Fanuc TP program (LS listing): hs0301h80_3.ls

/PROG  hs0301h80_3
/ATTR
COMMENT	= "19-03-01 11:47:14";
PROG_SIZE	= 0;
DEFAULT_GROUP	= 1, *, *, *, *;
/APPL
    ARC Welding Equipment: 1, *, *, *, *;
/MN
   1:  CALL HOME_ALL;
   1:  UFRAME_NUM = 1;
   1:  UTOOL_NUM = 3;
   1:  COL GUARD ADJUST 150;
   1:  PR[91] = PR[90];
   1:  PR[91,1] = PR[90,1] + -0.293;
   1:  PR[91,2] = PR[90,2] + 23.494;
   1:  PR[91,3] = PR[90,3] + 60.085;
   1:  PR[92] = PR[91];
   1:  PR[92,3] = PR[92,3] + 50;
   1:J PR[92] 10% FINE;
   1:L PR[91] R[100]mm/sec CNT100;
   1:  CALL LASER_DRAHT_START;
   1:  PR[91,1] = PR[90,1] + -6.009;
   1:  PR[91,2] = PR[90,2] + 23.979;
   1:L PR[91] R[100]mm/sec CNT100;
   1:  PR[91,1] = PR[90,1] + -6.508;
   1:  PR[91,2] = PR[90,2] + 23.917;
   1:L PR[91] R[100]mm/sec CNT100;
   1:  PR[91,1] = PR[90,1] + -12.344;
   1:  PR[91,2] = PR[90,2] + 22.945;
   1:L PR[91] R[100]mm/sec CNT100;
   1:  PR[91,1] = PR[90,1] + -12.597;
   1:  PR[91,2] = PR[90,2] + 22.847;
   1:L PR[91] R[100]mm/sec CNT100;
   1:  PR[91,1] = PR[90,1] + -18.195;
   1:  PR[91,2] = PR[90,2] + 20.363;
   1:L PR[91] R[100]mm/sec CNT100;
   1:  PR[91,1] = PR[90,1] + -18.230;
   1:  PR[91,2] = PR[90,2] + 20.339;
   1:L PR[91] R[100]mm/sec CNT100;
   1:  PR[91,1] = PR[90,1] + -23.139;
   1:  PR[91,2] = PR[90,2] + 16.449;
   1:L PR[91] R[100]mm/sec CNT100;
   1:  PR[91,1] = PR[90,1] + -26.912;
   1:  PR[91,2] = PR[90,2] + 11.480;
   1:L PR[91] R[100]mm/sec CNT100;
   1:  PR[91,1] = PR[90,1] + -29.270;
   1:  PR[91,2] = PR[90,2] + 5.788;
   1:L PR[91] R[100]mm/sec CNT100;
   1:  PR[91,1] = PR[90,1] + -30.068;
   1:  PR[91,2] = PR[90,2] + -0.337;
   1:L PR[91] R[100]mm/sec CNT100;
   1:  PR[91,1] = PR[90,1] + -30.060;
   1:  PR[91,2] = PR[90,2] + -0.419;
   1:L PR[91] R[100]mm/sec CNT100;
   1:  PR[91,1] = PR[90,1] + -29.269;
   1:  PR[91,2] = PR[90,2] + -6.417;
   1:L PR[91] R[100]mm/sec CNT100;
   1:  PR[91,1] = PR[90,1] + -26.906;
   1:  PR[91,2] = PR[90,2] + -12.115;
   1:L PR[91] R[100]mm/sec CNT100;
   1:  PR[91,1] = PR[90,1] + -23.137;
   1:  PR[91,2] = PR[90,2] + -17.075;
   1:L PR[91] R[100]mm/sec CNT100;
   1:  PR[91,1] = PR[90,1] + -18.184;
   1:  PR[91,2] = PR[90,2] + -20.996;
   1:L PR[91] R[100]mm/sec CNT100;
   1:  PR[91,1] = PR[90,1] + -12.564;
   1:  PR[91,2] = PR[90,2] + -23.482;
   1:L PR[91] R[100]mm/sec CNT100;
   1:  PR[91,1] = PR[90,1] + -12.309;
   1:  PR[91,2] = PR[90,2] + -23.579;
   1:L PR[91] R[100]mm/sec CNT100;
   1:  PR[91,1] = PR[90,1] + -6.470;
   1:  PR[91,2] = PR[90,2] + -24.544;
   1:L PR[91] R[100]mm/sec CNT100;
   1:  PR[91,1] = PR[90,1] + -5.966;
   1:  PR[91,2] = PR[90,2] + -24.604;
   1:L PR[91] R[100]mm/sec CNT100;
   1:  PR[91,1] = PR[90,1] + -0.295;
   1:  PR[91,2] = PR[90,2] + -24.113;
   1:L PR[91] R[100]mm/sec CNT100;
   1:  PR[91,1] = PR[90,1] + 0.454;
   1:  PR[91,2] = PR[90,2] + -24.114;
   1:L PR[91] R[100]mm/sec CNT100;
   1:  PR[91,1] = PR[90,1] + 5.405;
   1:  PR[91,2] = PR[90,2] + -24.549;
   1:L PR[91] R[100]mm/sec CNT100;
   1:  PR[91,1] = PR[90,1] + 6.160;
   1:  PR[91,2] = PR[90,2] + -24.608;
   1:L PR[91] R[100]mm/sec CNT100;
   1:  PR[91,1] = PR[90,1] + 6.349;
   1:  PR[91,2] = PR[90,2] + -24.596;
   1:L PR[91] R[100]mm/sec CNT100;
   1:  PR[91,1] = PR[90,1] + 12.478;
   1:  PR[91,2] = PR[90,2] + -23.575;
   1:L PR[91] R[100]mm/sec CNT100;
   1:  PR[91,1] = PR[90,1] + 12.730;
   1:  PR[91,2] = PR[90,2] + -23.477;
   1:L PR[91] R[100]mm/sec CNT100;
   1:  PR[91,1] = PR[90,1] + 18.333;
   1:  PR[91,2] = PR[90,2] + -20.999;
   1:L PR[91] R[100]mm/sec CNT100;
   1:  PR[91,1] = PR[90,1] + 18.368;
   1:  PR[91,2] = PR[90,2] + -20.974;
   1:L PR[91] R[100]mm/sec CNT100;
   1:  PR[91,1] = PR[90,1] + 23.284;
   1:  PR[91,2] = PR[90,2] + -17.085;
   1:L PR[91] R[100]mm/sec CNT100;
   1:  PR[91,1] = PR[90,1] + 27.064;
   1:  PR[91,2] = PR[90,2] + -12.111;
   1:L PR[91] R[100]mm/sec CNT100;
   1:  PR[91,1] = PR[90,1] + 29.425;
   1:  PR[91,2] = PR[90,2] + -6.423;
   1:L PR[91] R[100]mm/sec CNT100;
   1:  PR[91,1] = PR[90,1] + 30.225;
   1:  PR[91,2] = PR[90,2] + -0.287;
   1:L PR[91] R[100]mm/sec CNT100;
   1:  PR[91,1] = PR[90,1] + 30.217;
   1:  PR[91,2] = PR[90,2] + -0.204;
   1:L PR[91] R[100]mm/sec CNT100;
   1:  PR[91,1] = PR[90,1] + 29.427;
   1:  PR[91,2] = PR[90,2] + 5.793;
   1:L PR[91] R[100]mm/sec CNT100;
   1:  PR[91,1] = PR[90,1] + 27.069;
   1:  PR[91,2] = PR[90,2] + 11.477;
   1:L PR[91] R[100]mm/sec CNT100;
   1:  PR[91,1] = PR[90,1] + 23.297;
   1:  PR[91,2] = PR[90,2] + 16.449;
   1:L PR[91] R[100]mm/sec CNT100;
   1:  PR[91,1] = PR[90,1] + 18.388;
   1:  PR[91,2] = PR[90,2] + 20.339;
   1:L PR[91] R[100]mm/sec CNT100;
   1:  PR[91,1] = PR[90,1] + 18.353;
   1:  PR[91,2] = PR[90,2] + 20.363;
   1:L PR[91] R[100]mm/sec CNT100;
   1:  PR[91,1] = PR[90,1] + 12.755;
   1:  PR[91,2] = PR[90,2] + 22.846;
   1:L PR[91] R[100]mm/sec CNT100;
   1:  PR[91,1] = PR[90,1] + 12.502;
   1:  PR[91,2] = PR[90,2] + 22.944;
   1:L PR[91] R[100]mm/sec CNT100;
   1:  PR[91,1] = PR[90,1] + 6.667;
   1:  PR[91,2] = PR[90,2] + 23.917;
   1:L PR[91] R[100]mm/sec CNT100;
   1:  PR[91,1] = PR[90,1] + 6.167;
   1:  PR[91,2] = PR[90,2] + 23.979;
   1:L PR[91] R[100]mm/sec CNT100;
   1:  PR[91,1] = PR[90,1] + 0.451;
   1:  PR[91,2] = PR[90,2] + 23.494;
   1:L PR[91] R[100]mm/sec CNT100;
   1:  PR[91] = PR[90];
   1:  PR[91,1] = PR[90,1] + -0.281;
   1:  PR[91,2] = PR[90,2] + 23.657;
   1:  PR[91,3] = PR[90,3] + 60.695;
   1:L PR[91] R[100]mm/sec CNT100;
   1:  PR[91,1] = PR[90,1] + -3.910;
   1:  PR[91,2] = PR[90,2] + 23.972;
   1:L PR[91] R[100]mm/sec CNT100;
   1:  PR[91,1] = PR[90,1] + -5.747;
   1:  PR[91,2] = PR[90,2] + 24.117;
   1:L PR[91] R[100]mm/sec CNT100;
   1:  PR[91,1] = PR[90,1] + -6.520;
   1:  PR[91,2] = PR[90,2] + 24.021;
   1:L PR[91] R[100]mm/sec CNT100;
   1:  PR[91,1] = PR[90,1] + -12.103;
   1:  PR[91,2] = PR[90,2] + 23.091;
   1:L PR[91] R[100]mm/sec CNT100;
   1:  PR[91,1] = PR[90,1] + -12.618;
   1:  PR[91,2] = PR[90,2] + 22.891;
   1:L PR[91] R[100]mm/sec CNT100;
   1:  PR[91,1] = PR[90,1] + -17.973;
   1:  PR[91,2] = PR[90,2] + 20.516;
   1:L PR[91] R[100]mm/sec CNT100;
   1:  PR[91,1] = PR[90,1] + -18.245;
   1:  PR[91,2] = PR[90,2] + 20.323;
   1:L PR[91] R[100]mm/sec CNT100;
   1:  PR[91,1] = PR[90,1] + -22.986;
   1:  PR[91,2] = PR[90,2] + 16.568;
   1:L PR[91] R[100]mm/sec CNT100;
   1:  PR[91,1] = PR[90,1] + -23.039;
   1:  PR[91,2] = PR[90,2] + 16.508;
   1:L PR[91] R[100]mm/sec CNT100;
   1:  PR[91,1] = PR[90,1] + -26.772;
   1:  PR[91,2] = PR[90,2] + 11.549;
   1:L PR[91] R[100]mm/sec CNT100;
   1:  PR[91,1] = PR[90,1] + -29.127;
   1:  PR[91,2] = PR[90,2] + 5.807;
   1:L PR[91] R[100]mm/sec CNT100;
   1:  PR[91,1] = PR[90,1] + -29.691;
   1:  PR[91,2] = PR[90,2] + 1.477;
   1:L PR[91] R[100]mm/sec CNT100;
   1:  PR[91,1] = PR[90,1] + -29.926;
   1:  PR[91,2] = PR[90,2] + -0.313;
   1:L PR[91] R[100]mm/sec CNT100;
   1:  PR[91,1] = PR[90,1] + -29.126;
   1:  PR[91,2] = PR[90,2] + -6.434;
   1:L PR[91] R[100]mm/sec CNT100;
   1:  PR[91,1] = PR[90,1] + -26.767;
   1:  PR[91,2] = PR[90,2] + -12.181;
   1:L PR[91] R[100]mm/sec CNT100;
   1:  PR[91,1] = PR[90,1] + -23.035;
   1:  PR[91,2] = PR[90,2] + -17.133;
   1:L PR[91] R[100]mm/sec CNT100;
   1:  PR[91,1] = PR[90,1] + -22.969;
   1:  PR[91,2] = PR[90,2] + -17.208;
   1:L PR[91] R[100]mm/sec CNT100;
   1:  PR[91,1] = PR[90,1] + -18.054;
   1:  PR[91,2] = PR[90,2] + -21.096;
   1:L PR[91] R[100]mm/sec CNT100;
   1:  PR[91,1] = PR[90,1] + -17.983;
   1:  PR[91,2] = PR[90,2] + -21.140;
   1:L PR[91] R[100]mm/sec CNT100;
   1:  PR[91,1] = PR[90,1] + -12.579;
   1:  PR[91,2] = PR[90,2] + -23.531;
   1:L PR[91] R[100]mm/sec CNT100;
   1:  PR[91,1] = PR[90,1] + -12.060;
   1:  PR[91,2] = PR[90,2] + -23.726;
   1:L PR[91] R[100]mm/sec CNT100;
   1:  PR[91,1] = PR[90,1] + -6.479;
   1:  PR[91,2] = PR[90,2] + -24.649;
   1:L PR[91] R[100]mm/sec CNT100;
   1:  PR[91,1] = PR[90,1] + -5.703;
   1:  PR[91,2] = PR[90,2] + -24.741;
   1:L PR[91] R[100]mm/sec CNT100;
   1:  PR[91,1] = PR[90,1] + -0.280;
   1:  PR[91,2] = PR[90,2] + -24.276;
   1:L PR[91] R[100]mm/sec CNT100;
   1:  PR[91,1] = PR[90,1] + 0.438;
   1:L PR[91] R[100]mm/sec CNT100;
   1:  PR[91,1] = PR[90,1] + 5.904;
   1:  PR[91,2] = PR[90,2] + -24.744;
   1:L PR[91] R[100]mm/sec CNT100;
   1:  PR[91,1] = PR[90,1] + 6.232;
   1:  PR[91,2] = PR[90,2] + -24.725;
   1:L PR[91] R[100]mm/sec CNT100;
   1:  PR[91,1] = PR[90,1] + 11.997;
   1:  PR[91,2] = PR[90,2] + -23.769;
   1:L PR[91] R[100]mm/sec CNT100;
   1:  PR[91,1] = PR[90,1] + 12.226;
   1:  PR[91,2] = PR[90,2] + -23.725;
   1:L PR[91] R[100]mm/sec CNT100;
   1:  PR[91,1] = PR[90,1] + 12.754;
   1:  PR[91,2] = PR[90,2] + -23.520;
   1:L PR[91] R[100]mm/sec CNT100;
   1:  PR[91,1] = PR[90,1] + 18.112;
   1:  PR[91,2] = PR[90,2] + -21.151;
   1:L PR[91] R[100]mm/sec CNT100;
   1:  PR[91,1] = PR[90,1] + 18.385;
   1:  PR[91,2] = PR[90,2] + -20.958;
   1:L PR[91] R[100]mm/sec CNT100;
   1:  PR[91,1] = PR[90,1] + 23.131;
   1:  PR[91,2] = PR[90,2] + -17.203;
   1:L PR[91] R[100]mm/sec CNT100;
   1:  PR[91,1] = PR[90,1] + 23.184;
   1:  PR[91,2] = PR[90,2] + -17.144;
   1:L PR[91] R[100]mm/sec CNT100;
   1:  PR[91,1] = PR[90,1] + 26.923;
   1:  PR[91,2] = PR[90,2] + -12.181;
   1:L PR[91] R[100]mm/sec CNT100;
   1:  PR[91,1] = PR[90,1] + 29.283;
   1:  PR[91,2] = PR[90,2] + -6.442;
   1:L PR[91] R[100]mm/sec CNT100;
   1:  PR[91,1] = PR[90,1] + 30.083;
   1:  PR[91,2] = PR[90,2] + -0.312;
   1:L PR[91] R[100]mm/sec CNT100;
   1:  PR[91,1] = PR[90,1] + 29.285;
   1:  PR[91,2] = PR[90,2] + 5.810;
   1:L PR[91] R[100]mm/sec CNT100;
   1:  PR[91,1] = PR[90,1] + 26.930;
   1:  PR[91,2] = PR[90,2] + 11.544;
   1:L PR[91] R[100]mm/sec CNT100;
   1:  PR[91,1] = PR[90,1] + 23.204;
   1:  PR[91,2] = PR[90,2] + 16.496;
   1:L PR[91] R[100]mm/sec CNT100;
   1:  PR[91,1] = PR[90,1] + 23.139;
   1:  PR[91,2] = PR[90,2] + 16.570;
   1:L PR[91] R[100]mm/sec CNT100;
   1:  PR[91,1] = PR[90,1] + 18.403;
   1:  PR[91,2] = PR[90,2] + 20.323;
   1:L PR[91] R[100]mm/sec CNT100;
   1:  PR[91,1] = PR[90,1] + 18.131;
   1:  PR[91,2] = PR[90,2] + 20.516;
   1:L PR[91] R[100]mm/sec CNT100;
   1:  PR[91,1] = PR[90,1] + 12.776;
   1:  PR[91,2] = PR[90,2] + 22.891;
   1:L PR[91] R[100]mm/sec CNT100;
   1:  PR[91,1] = PR[90,1] + 12.261;
   1:  PR[91,2] = PR[90,2] + 23.090;
   1:L PR[91] R[100]mm/sec CNT100;
   1:  PR[91,1] = PR[90,1] + 6.678;
   1:  PR[91,2] = PR[90,2] + 24.021;
   1:L PR[91] R[100]mm/sec CNT100;
   1:  PR[91,1] = PR[90,1] + 5.905;
   1:  PR[91,2] = PR[90,2] + 24.117;
   1:L PR[91] R[100]mm/sec CNT100;
   1:  PR[91,1] = PR[90,1] + 4.068;
   1:  PR[91,2] = PR[90,2] + 23.972;
   1:L PR[91] R[100]mm/sec CNT100;
   1:  PR[91,1] = PR[90,1] + 0.438;
   1:  PR[91,2] = PR[90,2] + 23.657;
   1:L PR[91] R[100]mm/sec CNT100;
   1:  PR[91] = PR[90];
   1:  PR[91,1] = PR[90,1] + -0.266;
   1:  PR[91,2] = PR[90,2] + 23.820;
   1:  PR[91,3] = PR[90,3] + 61.305;
   1:L PR[91] R[100]mm/sec CNT100;
   1:  PR[91,1] = PR[90,1] + -3.087;
   1:  PR[91,2] = PR[90,2] + 24.065;
   1:L PR[91] R[100]mm/sec CNT100;
   1:  PR[91,1] = PR[90,1] + -5.489;
   1:  PR[91,2] = PR[90,2] + 24.255;
   1:L PR[91] R[100]mm/sec CNT100;
   1:  PR[91,1] = PR[90,1] + -6.532;
   1:  PR[91,2] = PR[90,2] + 24.126;
   1:L PR[91] R[100]mm/sec CNT100;
   1:  PR[91,1] = PR[90,1] + -11.861;
   1:  PR[91,2] = PR[90,2] + 23.237;
   1:L PR[91] R[100]mm/sec CNT100;
   1:  PR[91,1] = PR[90,1] + -12.639;
   1:  PR[91,2] = PR[90,2] + 22.936;
   1:L PR[91] R[100]mm/sec CNT100;
   1:  PR[91,1] = PR[90,1] + -17.751;
   1:  PR[91,2] = PR[90,2] + 20.668;
   1:L PR[91] R[100]mm/sec CNT100;
   1:  PR[91,1] = PR[90,1] + -18.261;
   1:  PR[91,2] = PR[90,2] + 20.307;
   1:L PR[91] R[100]mm/sec CNT100;
   1:  PR[91,1] = PR[90,1] + -22.787;
   1:  PR[91,2] = PR[90,2] + 16.722;
   1:L PR[91] R[100]mm/sec CNT100;
   1:  PR[91,1] = PR[90,1] + -23.006;
   1:  PR[91,2] = PR[90,2] + 16.476;
   1:L PR[91] R[100]mm/sec CNT100;
   1:  PR[91,1] = PR[90,1] + -26.589;
   1:  PR[91,2] = PR[90,2] + 11.717;
   1:L PR[91] R[100]mm/sec CNT100;
   1:  PR[91,1] = PR[90,1] + -26.683;
   1:  PR[91,2] = PR[90,2] + 11.554;
   1:L PR[91] R[100]mm/sec CNT100;
   1:  PR[91,1] = PR[90,1] + -28.980;
   1:  PR[91,2] = PR[90,2] + 5.964;
   1:L PR[91] R[100]mm/sec CNT100;
   1:  PR[91,1] = PR[90,1] + -29.019;
   1:  PR[91,2] = PR[90,2] + 5.848;
   1:L PR[91] R[100]mm/sec CNT100;
   1:  PR[91,1] = PR[90,1] + -29.815;
   1:  PR[91,2] = PR[90,2] + -0.312;
   1:L PR[91] R[100]mm/sec CNT100;
   1:  PR[91,1] = PR[90,1] + -29.020;
   1:  PR[91,2] = PR[90,2] + -6.471;
   1:L PR[91] R[100]mm/sec CNT100;
   1:  PR[91,1] = PR[90,1] + -28.986;
   1:  PR[91,2] = PR[90,2] + -6.576;
   1:L PR[91] R[100]mm/sec CNT100;
   1:  PR[91,1] = PR[90,1] + -26.690;
   1:  PR[91,2] = PR[90,2] + -12.163;
   1:L PR[91] R[100]mm/sec CNT100;
   1:  PR[91,1] = PR[90,1] + -26.592;
   1:  PR[91,2] = PR[90,2] + -12.338;
   1:L PR[91] R[100]mm/sec CNT100;
   1:  PR[91,1] = PR[90,1] + -23.014;
   1:  PR[91,2] = PR[90,2] + -17.084;
   1:L PR[91] R[100]mm/sec CNT100;
   1:  PR[91,1] = PR[90,1] + -22.771;
   1:  PR[91,2] = PR[90,2] + -17.361;
   1:L PR[91] R[100]mm/sec CNT100;
   1:  PR[91,1] = PR[90,1] + -17.951;
   1:  PR[91,2] = PR[90,2] + -21.175;
   1:L PR[91] R[100]mm/sec CNT100;
   1:  PR[91,1] = PR[90,1] + -17.752;
   1:  PR[91,2] = PR[90,2] + -21.296;
   1:L PR[91] R[100]mm/sec CNT100;
   1:  PR[91,1] = PR[90,1] + -12.593;
   1:  PR[91,2] = PR[90,2] + -23.579;
   1:L PR[91] R[100]mm/sec CNT100;
   1:  PR[91,1] = PR[90,1] + -11.812;
   1:  PR[91,2] = PR[90,2] + -23.874;
   1:L PR[91] R[100]mm/sec CNT100;
   1:  PR[91,1] = PR[90,1] + -6.489;
   1:  PR[91,2] = PR[90,2] + -24.754;
   1:L PR[91] R[100]mm/sec CNT100;
   1:  PR[91,1] = PR[90,1] + -5.435;
   1:  PR[91,2] = PR[90,2] + -24.879;
   1:L PR[91] R[100]mm/sec CNT100;
   1:  PR[91,1] = PR[90,1] + -4.039;
   1:  PR[91,2] = PR[90,2] + -24.770;
   1:L PR[91] R[100]mm/sec CNT100;
   1:  PR[91,1] = PR[90,1] + -0.268;
   1:  PR[91,2] = PR[90,2] + -24.438;
   1:L PR[91] R[100]mm/sec CNT100;
   1:  PR[91,1] = PR[90,1] + 0.425;
   1:L PR[91] R[100]mm/sec CNT100;
   1:  PR[91,1] = PR[90,1] + 4.197;
   1:  PR[91,2] = PR[90,2] + -24.770;
   1:L PR[91] R[100]mm/sec CNT100;
   1:  PR[91,1] = PR[90,1] + 5.636;
   1:  PR[91,2] = PR[90,2] + -24.882;
   1:L PR[91] R[100]mm/sec CNT100;
   1:  PR[91,1] = PR[90,1] + 6.114;
   1:  PR[91,2] = PR[90,2] + -24.853;
   1:L PR[91] R[100]mm/sec CNT100;
   1:  PR[91,1] = PR[90,1] + 11.615;
   1:  PR[91,2] = PR[90,2] + -23.941;
   1:L PR[91] R[100]mm/sec CNT100;
   1:  PR[91,1] = PR[90,1] + 11.989;
   1:  PR[91,2] = PR[90,2] + -23.870;
   1:L PR[91] R[100]mm/sec CNT100;
   1:  PR[91,1] = PR[90,1] + 12.777;
   1:  PR[91,2] = PR[90,2] + -23.564;
   1:L PR[91] R[100]mm/sec CNT100;
   1:  PR[91,1] = PR[90,1] + 17.890;
   1:  PR[91,2] = PR[90,2] + -21.303;
   1:L PR[91] R[100]mm/sec CNT100;
   1:  PR[91,1] = PR[90,1] + 18.401;
   1:  PR[91,2] = PR[90,2] + -20.941;
   1:L PR[91] R[100]mm/sec CNT100;
   1:  PR[91,1] = PR[90,1] + 22.933;
   1:  PR[91,2] = PR[90,2] + -17.357;
   1:L PR[91] R[100]mm/sec CNT100;
   1:  PR[91,1] = PR[90,1] + 23.152;
   1:  PR[91,2] = PR[90,2] + -17.111;
   1:L PR[91] R[100]mm/sec CNT100;
   1:  PR[91,1] = PR[90,1] + 26.740;
   1:  PR[91,2] = PR[90,2] + -12.348;
   1:L PR[91] R[100]mm/sec CNT100;
   1:  PR[91,1] = PR[90,1] + 26.835;
   1:  PR[91,2] = PR[90,2] + -12.185;
   1:L PR[91] R[100]mm/sec CNT100;
   1:  PR[91,1] = PR[90,1] + 29.135;
   1:  PR[91,2] = PR[90,2] + -6.598;
   1:L PR[91] R[100]mm/sec CNT100;
   1:  PR[91,1] = PR[90,1] + 29.174;
   1:  PR[91,2] = PR[90,2] + -6.482;
   1:L PR[91] R[100]mm/sec CNT100;
   1:  PR[91,1] = PR[90,1] + 29.965;
   1:  PR[91,2] = PR[90,2] + -0.403;
   1:L PR[91] R[100]mm/sec CNT100;
   1:  PR[91,1] = PR[90,1] + 29.974;
   1:  PR[91,2] = PR[90,2] + -0.325;
   1:L PR[91] R[100]mm/sec CNT100;
   1:  PR[91,1] = PR[90,1] + 29.178;
   1:  PR[91,2] = PR[90,2] + 5.846;
   1:L PR[91] R[100]mm/sec CNT100;
   1:  PR[91,1] = PR[90,1] + 29.145;
   1:  PR[91,2] = PR[90,2] + 5.951;
   1:L PR[91] R[100]mm/sec CNT100;
   1:  PR[91,1] = PR[90,1] + 26.852;
   1:  PR[91,2] = PR[90,2] + 11.526;
   1:L PR[91] R[100]mm/sec CNT100;
   1:  PR[91,1] = PR[90,1] + 26.754;
   1:  PR[91,2] = PR[90,2] + 11.701;
   1:L PR[91] R[100]mm/sec CNT100;
   1:  PR[91,1] = PR[90,1] + 23.183;
   1:  PR[91,2] = PR[90,2] + 16.448;
   1:L PR[91] R[100]mm/sec CNT100;
   1:  PR[91,1] = PR[90,1] + 22.940;
   1:  PR[91,2] = PR[90,2] + 16.724;
   1:L PR[91] R[100]mm/sec CNT100;
   1:  PR[91,1] = PR[90,1] + 18.419;
   1:  PR[91,2] = PR[90,2] + 20.307;
   1:L PR[91] R[100]mm/sec CNT100;
   1:  PR[91,1] = PR[90,1] + 17.909;
   1:  PR[91,2] = PR[90,2] + 20.668;
   1:L PR[91] R[100]mm/sec CNT100;
   1:  PR[91,1] = PR[90,1] + 12.797;
   1:  PR[91,2] = PR[90,2] + 22.935;
   1:L PR[91] R[100]mm/sec CNT100;
   1:  PR[91,1] = PR[90,1] + 12.019;
   1:  PR[91,2] = PR[90,2] + 23.237;
   1:L PR[91] R[100]mm/sec CNT100;
   1:  PR[91,1] = PR[90,1] + 6.690;
   1:  PR[91,2] = PR[90,2] + 24.126;
   1:L PR[91] R[100]mm/sec CNT100;
   1:  PR[91,1] = PR[90,1] + 5.647;
   1:  PR[91,2] = PR[90,2] + 24.255;
   1:L PR[91] R[100]mm/sec CNT100;
   1:  PR[91,1] = PR[90,1] + 3.244;
   1:  PR[91,2] = PR[90,2] + 24.065;
   1:L PR[91] R[100]mm/sec CNT100;
   1:  PR[91,1] = PR[90,1] + 0.424;
   1:  PR[91,2] = PR[90,2] + 23.820;
   1:L PR[91] R[100]mm/sec CNT100;
   1:  PR[91] = PR[90];
   1:  PR[91,1] = PR[90,1] + -0.249;
   1:  PR[91,2] = PR[90,2] + 23.984;
   1:  PR[91,3] = PR[90,3] + 61.915;
   1:L PR[91] R[100]mm/sec CNT100;
   1:  PR[91,1] = PR[90,1] + -5.233;
   1:  PR[91,2] = PR[90,2] + 24.392;
   1:L PR[91] R[100]mm/sec CNT100;
   1:  PR[91,1] = PR[90,1] + -6.544;
   1:  PR[91,2] = PR[90,2] + 24.230;
   1:L PR[91] R[100]mm/sec CNT100;
   1:  PR[91,1] = PR[90,1] + -11.619;
   1:  PR[91,2] = PR[90,2] + 23.384;
   1:L PR[91] R[100]mm/sec CNT100;
   1:  PR[91,1] = PR[90,1] + -12.660;
   1:  PR[91,2] = PR[90,2] + 22.981;
   1:L PR[91] R[100]mm/sec CNT100;
   1:  PR[91,1] = PR[90,1] + -17.529;
   1:  PR[91,2] = PR[90,2] + 20.821;
   1:L PR[91] R[100]mm/sec CNT100;
   1:  PR[91,1] = PR[90,1] + -18.277;
   1:  PR[91,2] = PR[90,2] + 20.291;
   1:L PR[91] R[100]mm/sec CNT100;
   1:  PR[91,1] = PR[90,1] + -22.588;
   1:  PR[91,2] = PR[90,2] + 16.876;
   1:L PR[91] R[100]mm/sec CNT100;
   1:  PR[91,1] = PR[90,1] + -22.974;
   1:  PR[91,2] = PR[90,2] + 16.443;
   1:L PR[91] R[100]mm/sec CNT100;
   1:  PR[91,1] = PR[90,1] + -26.386;
   1:  PR[91,2] = PR[90,2] + 11.910;
   1:L PR[91] R[100]mm/sec CNT100;
   1:  PR[91,1] = PR[90,1] + -26.605;
   1:  PR[91,2] = PR[90,2] + 11.534;
   1:L PR[91] R[100]mm/sec CNT100;
   1:  PR[91,1] = PR[90,1] + -28.792;
   1:  PR[91,2] = PR[90,2] + 6.211;
   1:L PR[91] R[100]mm/sec CNT100;
   1:  PR[91,1] = PR[90,1] + -28.917;
   1:  PR[91,2] = PR[90,2] + 5.841;
   1:L PR[91] R[100]mm/sec CNT100;
   1:  PR[91,1] = PR[90,1] + -29.707;
   1:  PR[91,2] = PR[90,2] + -0.311;
   1:L PR[91] R[100]mm/sec CNT100;
   1:  PR[91,1] = PR[90,1] + -28.963;
   1:  PR[91,2] = PR[90,2] + -6.019;
   1:L PR[91] R[100]mm/sec CNT100;
   1:  PR[91,1] = PR[90,1] + -28.916;
   1:  PR[91,2] = PR[90,2] + -6.465;
   1:L PR[91] R[100]mm/sec CNT100;
   1:  PR[91,1] = PR[90,1] + -28.810;
   1:  PR[91,2] = PR[90,2] + -6.797;
   1:L PR[91] R[100]mm/sec CNT100;
   1:  PR[91,1] = PR[90,1] + -26.623;
   1:  PR[91,2] = PR[90,2] + -12.117;
   1:L PR[91] R[100]mm/sec CNT100;
   1:  PR[91,1] = PR[90,1] + -26.401;
   1:  PR[91,2] = PR[90,2] + -12.515;
   1:L PR[91] R[100]mm/sec CNT100;
   1:  PR[91,1] = PR[90,1] + -22.993;
   1:  PR[91,2] = PR[90,2] + -17.036;
   1:L PR[91] R[100]mm/sec CNT100;
   1:  PR[91,1] = PR[90,1] + -22.572;
   1:  PR[91,2] = PR[90,2] + -17.515;
   1:L PR[91] R[100]mm/sec CNT100;
   1:  PR[91,1] = PR[90,1] + -17.849;
   1:  PR[91,2] = PR[90,2] + -21.254;
   1:L PR[91] R[100]mm/sec CNT100;
   1:  PR[91,1] = PR[90,1] + -17.521;
   1:  PR[91,2] = PR[90,2] + -21.453;
   1:L PR[91] R[100]mm/sec CNT100;
   1:  PR[91,1] = PR[90,1] + -12.608;
   1:  PR[91,2] = PR[90,2] + -23.627;
   1:L PR[91] R[100]mm/sec CNT100;
   1:  PR[91,1] = PR[90,1] + -11.563;
   1:  PR[91,2] = PR[90,2] + -24.022;
   1:L PR[91] R[100]mm/sec CNT100;
   1:  PR[91,1] = PR[90,1] + -6.498;
   1:  PR[91,2] = PR[90,2] + -24.860;
   1:L PR[91] R[100]mm/sec CNT100;
   1:  PR[91,1] = PR[90,1] + -5.173;
   1:  PR[91,2] = PR[90,2] + -25.016;
   1:L PR[91] R[100]mm/sec CNT100;
   1:  PR[91,1] = PR[90,1] + -3.435;
   1:  PR[91,2] = PR[90,2] + -24.881;
   1:L PR[91] R[100]mm/sec CNT100;
   1:  PR[91,1] = PR[90,1] + -0.254;
   1:  PR[91,2] = PR[90,2] + -24.601;
   1:L PR[91] R[100]mm/sec CNT100;
   1:  PR[91,1] = PR[90,1] + 0.411;
   1:L PR[91] R[100]mm/sec CNT100;
   1:  PR[91,1] = PR[90,1] + 3.593;
   1:  PR[91,2] = PR[90,2] + -24.881;
   1:L PR[91] R[100]mm/sec CNT100;
   1:  PR[91,1] = PR[90,1] + 5.374;
   1:  PR[91,2] = PR[90,2] + -25.019;
   1:L PR[91] R[100]mm/sec CNT100;
   1:  PR[91,1] = PR[90,1] + 5.996;
   1:  PR[91,2] = PR[90,2] + -24.982;
   1:L PR[91] R[100]mm/sec CNT100;
   1:  PR[91,1] = PR[90,1] + 11.234;
   1:  PR[91,2] = PR[90,2] + -24.113;
   1:L PR[91] R[100]mm/sec CNT100;
   1:  PR[91,1] = PR[90,1] + 11.751;
   1:  PR[91,2] = PR[90,2] + -24.015;
   1:L PR[91] R[100]mm/sec CNT100;
   1:  PR[91,1] = PR[90,1] + 12.800;
   1:  PR[91,2] = PR[90,2] + -23.607;
   1:L PR[91] R[100]mm/sec CNT100;
   1:  PR[91,1] = PR[90,1] + 17.668;
   1:  PR[91,2] = PR[90,2] + -21.455;
   1:L PR[91] R[100]mm/sec CNT100;
   1:  PR[91,1] = PR[90,1] + 18.417;
   1:  PR[91,2] = PR[90,2] + -20.925;
   1:L PR[91] R[100]mm/sec CNT100;
   1:  PR[91,1] = PR[90,1] + 22.734;
   1:  PR[91,2] = PR[90,2] + -17.510;
   1:L PR[91] R[100]mm/sec CNT100;
   1:  PR[91,1] = PR[90,1] + 23.121;
   1:  PR[91,2] = PR[90,2] + -17.077;
   1:L PR[91] R[100]mm/sec CNT100;
   1:  PR[91,1] = PR[90,1] + 26.538;
   1:  PR[91,2] = PR[90,2] + -12.541;
   1:L PR[91] R[100]mm/sec CNT100;
   1:  PR[91,1] = PR[90,1] + 26.757;
   1:  PR[91,2] = PR[90,2] + -12.165;
   1:L PR[91] R[100]mm/sec CNT100;
   1:  PR[91,1] = PR[90,1] + 28.948;
   1:  PR[91,2] = PR[90,2] + -6.844;
   1:L PR[91] R[100]mm/sec CNT100;
   1:  PR[91,1] = PR[90,1] + 29.072;
   1:  PR[91,2] = PR[90,2] + -6.475;
   1:L PR[91] R[100]mm/sec CNT100;
   1:  PR[91,1] = PR[90,1] + 29.825;
   1:  PR[91,2] = PR[90,2] + -0.688;
   1:L PR[91] R[100]mm/sec CNT100;
   1:  PR[91,1] = PR[90,1] + 29.865;
   1:  PR[91,2] = PR[90,2] + -0.326;
   1:L PR[91] R[100]mm/sec CNT100;
   1:  PR[91,1] = PR[90,1] + 29.121;
   1:  PR[91,2] = PR[90,2] + 5.395;
   1:L PR[91] R[100]mm/sec CNT100;
   1:  PR[91,1] = PR[90,1] + 29.074;
   1:  PR[91,2] = PR[90,2] + 5.840;
   1:L PR[91] R[100]mm/sec CNT100;
   1:  PR[91,1] = PR[90,1] + 28.969;
   1:  PR[91,2] = PR[90,2] + 6.172;
   1:L PR[91] R[100]mm/sec CNT100;
   1:  PR[91,1] = PR[90,1] + 26.785;
   1:  PR[91,2] = PR[90,2] + 11.481;
   1:L PR[91] R[100]mm/sec CNT100;
   1:  PR[91,1] = PR[90,1] + 26.563;
   1:  PR[91,2] = PR[90,2] + 11.879;
   1:L PR[91] R[100]mm/sec CNT100;
   1:  PR[91,1] = PR[90,1] + 23.161;
   1:  PR[91,2] = PR[90,2] + 16.400;
   1:L PR[91] R[100]mm/sec CNT100;
   1:  PR[91,1] = PR[90,1] + 22.741;
   1:  PR[91,2] = PR[90,2] + 16.878;
   1:L PR[91] R[100]mm/sec CNT100;
   1:  PR[91,1] = PR[90,1] + 18.434;
   1:  PR[91,2] = PR[90,2] + 20.291;
   1:L PR[91] R[100]mm/sec CNT100;
   1:  PR[91,1] = PR[90,1] + 17.687;
   1:  PR[91,2] = PR[90,2] + 20.821;
   1:L PR[91] R[100]mm/sec CNT100;
   1:  PR[91,1] = PR[90,1] + 12.817;
   1:  PR[91,2] = PR[90,2] + 22.980;
   1:L PR[91] R[100]mm/sec CNT100;
   1:  PR[91,1] = PR[90,1] + 11.777;
   1:  PR[91,2] = PR[90,2] + 23.383;
   1:L PR[91] R[100]mm/sec CNT100;
   1:  PR[91,1] = PR[90,1] + 6.702;
   1:  PR[91,2] = PR[90,2] + 24.230;
   1:L PR[91] R[100]mm/sec CNT100;
   1:  PR[91,1] = PR[90,1] + 5.391;
   1:  PR[91,2] = PR[90,2] + 24.392;
   1:L PR[91] R[100]mm/sec CNT100;
   1:  PR[91,1] = PR[90,1] + 0.406;
   1:  PR[91,2] = PR[90,2] + 23.984;
   1:L PR[91] R[100]mm/sec CNT100;
   1:  PR[91] = PR[90];
   1:  PR[91,1] = PR[90,1] + -0.234;
   1:  PR[91,2] = PR[90,2] + 24.147;
   1:  PR[91,3] = PR[90,3] + 62.525;
   1:L PR[91] R[100]mm/sec CNT100;
   1:  PR[91,1] = PR[90,1] + -4.974;
   1:  PR[91,2] = PR[90,2] + 24.530;
   1:L PR[91] R[100]mm/sec CNT100;
   1:  PR[91,1] = PR[90,1] + -6.556;
   1:  PR[91,2] = PR[90,2] + 24.334;
   1:L PR[91] R[100]mm/sec CNT100;
   1:  PR[91,1] = PR[90,1] + -11.378;
   1:  PR[91,2] = PR[90,2] + 23.530;
   1:L PR[91] R[100]mm/sec CNT100;
   1:  PR[91,1] = PR[90,1] + -12.681;
   1:  PR[91,2] = PR[90,2] + 23.025;
   1:L PR[91] R[100]mm/sec CNT100;
   1:  PR[91,1] = PR[90,1] + -17.307;
   1:  PR[91,2] = PR[90,2] + 20.973;
   1:L PR[91] R[100]mm/sec CNT100;
   1:  PR[91,1] = PR[90,1] + -18.292;
   1:  PR[91,2] = PR[90,2] + 20.275;
   1:L PR[91] R[100]mm/sec CNT100;
   1:  PR[91,1] = PR[90,1] + -22.389;
   1:  PR[91,2] = PR[90,2] + 17.030;
   1:L PR[91] R[100]mm/sec CNT100;
   1:  PR[91,1] = PR[90,1] + -22.942;
   1:  PR[91,2] = PR[90,2] + 16.410;
   1:L PR[91] R[100]mm/sec CNT100;
   1:  PR[91,1] = PR[90,1] + -26.184;
   1:  PR[91,2] = PR[90,2] + 12.104;
   1:L PR[91] R[100]mm/sec CNT100;
   1:  PR[91,1] = PR[90,1] + -26.528;
   1:  PR[91,2] = PR[90,2] + 11.514;
   1:L PR[91] R[100]mm/sec CNT100;
   1:  PR[91,1] = PR[90,1] + -28.605;
   1:  PR[91,2] = PR[90,2] + 6.458;
   1:L PR[91] R[100]mm/sec CNT100;
   1:  PR[91,1] = PR[90,1] + -28.815;
   1:  PR[91,2] = PR[90,2] + 5.834;
   1:L PR[91] R[100]mm/sec CNT100;
   1:  PR[91,1] = PR[90,1] + -29.529;
   1:  PR[91,2] = PR[90,2] + 0.347;
   1:L PR[91] R[100]mm/sec CNT100;
   1:  PR[91,1] = PR[90,1] + -29.600;
   1:  PR[91,2] = PR[90,2] + -0.298;
   1:L PR[91] R[100]mm/sec CNT100;
   1:  PR[91,1] = PR[90,1] + -28.892;
   1:  PR[91,2] = PR[90,2] + -5.730;
   1:L PR[91] R[100]mm/sec CNT100;
   1:  PR[91,1] = PR[90,1] + -28.818;
   1:  PR[91,2] = PR[90,2] + -6.441;
   1:L PR[91] R[100]mm/sec CNT100;
   1:  PR[91,1] = PR[90,1] + -28.634;
   1:  PR[91,2] = PR[90,2] + -7.018;
   1:L PR[91] R[100]mm/sec CNT100;
   1:  PR[91,1] = PR[90,1] + -26.556;
   1:  PR[91,2] = PR[90,2] + -12.072;
   1:L PR[91] R[100]mm/sec CNT100;
   1:  PR[91,1] = PR[90,1] + -26.210;
   1:  PR[91,2] = PR[90,2] + -12.693;
   1:L PR[91] R[100]mm/sec CNT100;
   1:  PR[91,1] = PR[90,1] + -22.972;
   1:  PR[91,2] = PR[90,2] + -16.987;
   1:L PR[91] R[100]mm/sec CNT100;
   1:  PR[91,1] = PR[90,1] + -22.374;
   1:  PR[91,2] = PR[90,2] + -17.668;
   1:L PR[91] R[100]mm/sec CNT100;
   1:  PR[91,1] = PR[90,1] + -17.746;
   1:  PR[91,2] = PR[90,2] + -21.333;
   1:L PR[91] R[100]mm/sec CNT100;
   1:  PR[91,1] = PR[90,1] + -17.291;
   1:  PR[91,2] = PR[90,2] + -21.610;
   1:L PR[91] R[100]mm/sec CNT100;
   1:  PR[91,1] = PR[90,1] + -12.623;
   1:  PR[91,2] = PR[90,2] + -23.675;
   1:L PR[91] R[100]mm/sec CNT100;
   1:  PR[91,1] = PR[90,1] + -11.314;
   1:  PR[91,2] = PR[90,2] + -24.170;
   1:L PR[91] R[100]mm/sec CNT100;
   1:  PR[91,1] = PR[90,1] + -6.507;
   1:  PR[91,2] = PR[90,2] + -24.965;
   1:L PR[91] R[100]mm/sec CNT100;
   1:  PR[91,1] = PR[90,1] + -4.911;
   1:  PR[91,2] = PR[90,2] + -25.153;
   1:L PR[91] R[100]mm/sec CNT100;
   1:  PR[91,1] = PR[90,1] + -2.831;
   1:  PR[91,2] = PR[90,2] + -24.991;
   1:L PR[91] R[100]mm/sec CNT100;
   1:  PR[91,1] = PR[90,1] + -0.240;
   1:  PR[91,2] = PR[90,2] + -24.763;
   1:L PR[91] R[100]mm/sec CNT100;
   1:  PR[91,1] = PR[90,1] + 0.397;
   1:L PR[91] R[100]mm/sec CNT100;
   1:  PR[91,1] = PR[90,1] + 2.989;
   1:  PR[91,2] = PR[90,2] + -24.991;
   1:L PR[91] R[100]mm/sec CNT100;
   1:  PR[91,1] = PR[90,1] + 5.111;
   1:  PR[91,2] = PR[90,2] + -25.156;
   1:L PR[91] R[100]mm/sec CNT100;
   1:  PR[91,1] = PR[90,1] + 5.878;
   1:  PR[91,2] = PR[90,2] + -25.110;
   1:L PR[91] R[100]mm/sec CNT100;
   1:  PR[91,1] = PR[90,1] + 10.853;
   1:  PR[91,2] = PR[90,2] + -24.285;
   1:L PR[91] R[100]mm/sec CNT100;
   1:  PR[91,1] = PR[90,1] + 11.514;
   1:  PR[91,2] = PR[90,2] + -24.160;
   1:L PR[91] R[100]mm/sec CNT100;
   1:  PR[91,1] = PR[90,1] + 12.824;
   1:  PR[91,2] = PR[90,2] + -23.651;
   1:L PR[91] R[100]mm/sec CNT100;
   1:  PR[91,1] = PR[90,1] + 17.446;
   1:  PR[91,2] = PR[90,2] + -21.607;
   1:L PR[91] R[100]mm/sec CNT100;
   1:  PR[91,1] = PR[90,1] + 18.434;
   1:  PR[91,2] = PR[90,2] + -20.909;
   1:L PR[91] R[100]mm/sec CNT100;
   1:  PR[91,1] = PR[90,1] + 22.536;
   1:  PR[91,2] = PR[90,2] + -17.664;
   1:L PR[91] R[100]mm/sec CNT100;
   1:  PR[91,1] = PR[90,1] + 23.089;
   1:  PR[91,2] = PR[90,2] + -17.044;
   1:L PR[91] R[100]mm/sec CNT100;
   1:  PR[91,1] = PR[90,1] + 26.336;
   1:  PR[91,2] = PR[90,2] + -12.734;
   1:L PR[91] R[100]mm/sec CNT100;
   1:  PR[91,1] = PR[90,1] + 26.680;
   1:  PR[91,2] = PR[90,2] + -12.144;
   1:L PR[91] R[100]mm/sec CNT100;
   1:  PR[91,1] = PR[90,1] + 28.760;
   1:  PR[91,2] = PR[90,2] + -7.090;
   1:L PR[91] R[100]mm/sec CNT100;
   1:  PR[91,1] = PR[90,1] + 28.970;
   1:  PR[91,2] = PR[90,2] + -6.467;
   1:L PR[91] R[100]mm/sec CNT100;
   1:  PR[91,1] = PR[90,1] + 29.686;
   1:  PR[91,2] = PR[90,2] + -0.972;
   1:L PR[91] R[100]mm/sec CNT100;
   1:  PR[91,1] = PR[90,1] + 29.757;
   1:  PR[91,2] = PR[90,2] + -0.326;
   1:L PR[91] R[100]mm/sec CNT100;
   1:  PR[91,1] = PR[90,1] + 29.050;
   1:  PR[91,2] = PR[90,2] + 5.106;
   1:L PR[91] R[100]mm/sec CNT100;
   1:  PR[91,1] = PR[90,1] + 28.976;
   1:  PR[91,2] = PR[90,2] + 5.817;
   1:L PR[91] R[100]mm/sec CNT100;
   1:  PR[91,1] = PR[90,1] + 28.792;
   1:  PR[91,2] = PR[90,2] + 6.393;
   1:L PR[91] R[100]mm/sec CNT100;
   1:  PR[91,1] = PR[90,1] + 26.719;
   1:  PR[91,2] = PR[90,2] + 11.436;
   1:L PR[91] R[100]mm/sec CNT100;
   1:  PR[91,1] = PR[90,1] + 26.372;
   1:  PR[91,2] = PR[90,2] + 12.057;
   1:L PR[91] R[100]mm/sec CNT100;
   1:  PR[91,1] = PR[90,1] + 23.140;
   1:  PR[91,2] = PR[90,2] + 16.352;
   1:L PR[91] R[100]mm/sec CNT100;
   1:  PR[91,1] = PR[90,1] + 22.542;
   1:  PR[91,2] = PR[90,2] + 17.032;
   1:L PR[91] R[100]mm/sec CNT100;
   1:  PR[91,1] = PR[90,1] + 18.450;
   1:  PR[91,2] = PR[90,2] + 20.275;
   1:L PR[91] R[100]mm/sec CNT100;
   1:  PR[91,1] = PR[90,1] + 17.464;
   1:  PR[91,2] = PR[90,2] + 20.973;
   1:L PR[91] R[100]mm/sec CNT100;
   1:  PR[91,1] = PR[90,1] + 12.838;
   1:  PR[91,2] = PR[90,2] + 23.025;
   1:L PR[91] R[100]mm/sec CNT100;
   1:  PR[91,1] = PR[90,1] + 11.535;
   1:  PR[91,2] = PR[90,2] + 23.530;
   1:L PR[91] R[100]mm/sec CNT100;
   1:  PR[91,1] = PR[90,1] + 6.714;
   1:  PR[91,2] = PR[90,2] + 24.334;
   1:L PR[91] R[100]mm/sec CNT100;
   1:  PR[91,1] = PR[90,1] + 5.132;
   1:  PR[91,2] = PR[90,2] + 24.530;
   1:L PR[91] R[100]mm/sec CNT100;
   1:  PR[91,1] = PR[90,1] + 0.391;
   1:  PR[91,2] = PR[90,2] + 24.147;
   1:L PR[91] R[100]mm/sec CNT100;
   1:  PR[91] = PR[90];
   1:  PR[91,1] = PR[90,1] + -0.219;
   1:  PR[91,2] = PR[90,2] + 24.310;
   1:  PR[91,3] = PR[90,3] + 63.135;
   1:L PR[91] R[100]mm/sec CNT100;
   1:  PR[91,1] = PR[90,1] + -4.715;
   1:  PR[91,2] = PR[90,2] + 24.667;
   1:L PR[91] R[100]mm/sec CNT100;
   1:  PR[91,1] = PR[90,1] + -6.568;
   1:  PR[91,2] = PR[90,2] + 24.438;
   1:L PR[91] R[100]mm/sec CNT100;
   1:  PR[91,1] = PR[90,1] + -11.136;
   1:  PR[91,2] = PR[90,2] + 23.677;
   1:L PR[91] R[100]mm/sec CNT100;
   1:  PR[91,1] = PR[90,1] + -12.702;
   1:  PR[91,2] = PR[90,2] + 23.070;
   1:L PR[91] R[100]mm/sec CNT100;
   1:  PR[91,1] = PR[90,1] + -17.085;
   1:  PR[91,2] = PR[90,2] + 21.126;
   1:L PR[91] R[100]mm/sec CNT100;
   1:  PR[91,1] = PR[90,1] + -18.308;
   1:  PR[91,2] = PR[90,2] + 20.260;
   1:L PR[91] R[100]mm/sec CNT100;
   1:  PR[91,1] = PR[90,1] + -22.190;
   1:  PR[91,2] = PR[90,2] + 17.184;
   1:L PR[91] R[100]mm/sec CNT100;
   1:  PR[91,1] = PR[90,1] + -22.910;
   1:  PR[91,2] = PR[90,2] + 16.378;
   1:L PR[91] R[100]mm/sec CNT100;
   1:  PR[91,1] = PR[90,1] + -25.981;
   1:  PR[91,2] = PR[90,2] + 12.297;
   1:L PR[91] R[100]mm/sec CNT100;
   1:  PR[91,1] = PR[90,1] + -26.450;
   1:  PR[91,2] = PR[90,2] + 11.494;
   1:L PR[91] R[100]mm/sec CNT100;
   1:  PR[91,1] = PR[90,1] + -28.417;
   1:  PR[91,2] = PR[90,2] + 6.704;
   1:L PR[91] R[100]mm/sec CNT100;
   1:  PR[91,1] = PR[90,1] + -28.713;
   1:  PR[91,2] = PR[90,2] + 5.827;
   1:L PR[91] R[100]mm/sec CNT100;
   1:  PR[91,1] = PR[90,1] + -29.389;
   1:  PR[91,2] = PR[90,2] + 0.632;
   1:L PR[91] R[100]mm/sec CNT100;
   1:  PR[91,1] = PR[90,1] + -29.492;
   1:  PR[91,2] = PR[90,2] + -0.298;
   1:L PR[91] R[100]mm/sec CNT100;
   1:  PR[91,1] = PR[90,1] + -28.821;
   1:  PR[91,2] = PR[90,2] + -5.442;
   1:L PR[91] R[100]mm/sec CNT100;
   1:  PR[91,1] = PR[90,1] + -28.719;
   1:  PR[91,2] = PR[90,2] + -6.418;
   1:L PR[91] R[100]mm/sec CNT100;
   1:  PR[91,1] = PR[90,1] + -28.458;
   1:  PR[91,2] = PR[90,2] + -7.240;
   1:L PR[91] R[100]mm/sec CNT100;
   1:  PR[91,1] = PR[90,1] + -26.490;
   1:  PR[91,2] = PR[90,2] + -12.027;
   1:L PR[91] R[100]mm/sec CNT100;
   1:  PR[91,1] = PR[90,1] + -26.018;
   1:  PR[91,2] = PR[90,2] + -12.870;
   1:L PR[91] R[100]mm/sec CNT100;
   1:  PR[91,1] = PR[90,1] + -22.951;
   1:  PR[91,2] = PR[90,2] + -16.939;
   1:L PR[91] R[100]mm/sec CNT100;
   1:  PR[91,1] = PR[90,1] + -22.175;
   1:  PR[91,2] = PR[90,2] + -17.822;
   1:L PR[91] R[100]mm/sec CNT100;
   1:  PR[91,1] = PR[90,1] + -17.643;
   1:  PR[91,2] = PR[90,2] + -21.412;
   1:L PR[91] R[100]mm/sec CNT100;
   1:  PR[91,1] = PR[90,1] + -17.060;
   1:  PR[91,2] = PR[90,2] + -21.767;
   1:L PR[91] R[100]mm/sec CNT100;
   1:  PR[91,1] = PR[90,1] + -12.638;
   1:  PR[91,2] = PR[90,2] + -23.723;
   1:L PR[91] R[100]mm/sec CNT100;
   1:  PR[91,1] = PR[90,1] + -11.066;
   1:  PR[91,2] = PR[90,2] + -24.318;
   1:L PR[91] R[100]mm/sec CNT100;
   1:  PR[91,1] = PR[90,1] + -6.516;
   1:  PR[91,2] = PR[90,2] + -25.070;
   1:L PR[91] R[100]mm/sec CNT100;
   1:  PR[91,1] = PR[90,1] + -4.649;
   1:  PR[91,2] = PR[90,2] + -25.290;
   1:L PR[91] R[100]mm/sec CNT100;
   1:  PR[91,1] = PR[90,1] + -2.228;
   1:  PR[91,2] = PR[90,2] + -25.102;
   1:L PR[91] R[100]mm/sec CNT100;
   1:  PR[91,1] = PR[90,1] + -0.225;
   1:  PR[91,2] = PR[90,2] + -24.926;
   1:L PR[91] R[100]mm/sec CNT100;
   1:  PR[91,1] = PR[90,1] + 0.383;
   1:L PR[91] R[100]mm/sec CNT100;
   1:  PR[91,1] = PR[90,1] + 2.386;
   1:  PR[91,2] = PR[90,2] + -25.102;
   1:L PR[91] R[100]mm/sec CNT100;
   1:  PR[91,1] = PR[90,1] + 4.849;
   1:  PR[91,2] = PR[90,2] + -25.293;
   1:L PR[91] R[100]mm/sec CNT100;
   1:  PR[91,1] = PR[90,1] + 5.760;
   1:  PR[91,2] = PR[90,2] + -25.239;
   1:L PR[91] R[100]mm/sec CNT100;
   1:  PR[91,1] = PR[90,1] + 10.471;
   1:  PR[91,2] = PR[90,2] + -24.457;
   1:L PR[91] R[100]mm/sec CNT100;
   1:  PR[91,1] = PR[90,1] + 11.276;
   1:  PR[91,2] = PR[90,2] + -24.305;
   1:L PR[91] R[100]mm/sec CNT100;
   1:  PR[91,1] = PR[90,1] + 12.847;
   1:  PR[91,2] = PR[90,2] + -23.695;
   1:L PR[91] R[100]mm/sec CNT100;
   1:  PR[91,1] = PR[90,1] + 17.225;
   1:  PR[91,2] = PR[90,2] + -21.759;
   1:L PR[91] R[100]mm/sec CNT100;
   1:  PR[91,1] = PR[90,1] + 18.450;
   1:  PR[91,2] = PR[90,2] + -20.892;
   1:L PR[91] R[100]mm/sec CNT100;
   1:  PR[91,1] = PR[90,1] + 22.338;
   1:  PR[91,2] = PR[90,2] + -17.817;
   1:L PR[91] R[100]mm/sec CNT100;
   1:  PR[91,1] = PR[90,1] + 23.057;
   1:  PR[91,2] = PR[90,2] + -17.011;
   1:L PR[91] R[100]mm/sec CNT100;
   1:  PR[91,1] = PR[90,1] + 26.134;
   1:  PR[91,2] = PR[90,2] + -12.927;
   1:L PR[91] R[100]mm/sec CNT100;
   1:  PR[91,1] = PR[90,1] + 26.602;
   1:  PR[91,2] = PR[90,2] + -12.124;
   1:L PR[91] R[100]mm/sec CNT100;
   1:  PR[91,1] = PR[90,1] + 28.573;
   1:  PR[91,2] = PR[90,2] + -7.336;
   1:L PR[91] R[100]mm/sec CNT100;
   1:  PR[91,1] = PR[90,1] + 28.868;
   1:  PR[91,2] = PR[90,2] + -6.460;
   1:L PR[91] R[100]mm/sec CNT100;
   1:  PR[91,1] = PR[90,1] + 29.546;
   1:  PR[91,2] = PR[90,2] + -1.256;
   1:L PR[91] R[100]mm/sec CNT100;
   1:  PR[91,1] = PR[90,1] + 29.649;
   1:  PR[91,2] = PR[90,2] + -0.326;
   1:L PR[91] R[100]mm/sec CNT100;
   1:  PR[91,1] = PR[90,1] + 28.979;
   1:  PR[91,2] = PR[90,2] + 4.818;
   1:L PR[91] R[100]mm/sec CNT100;
   1:  PR[91,1] = PR[90,1] + 28.877;
   1:  PR[91,2] = PR[90,2] + 5.793;
   1:L PR[91] R[100]mm/sec CNT100;
   1:  PR[91,1] = PR[90,1] + 28.616;
   1:  PR[91,2] = PR[90,2] + 6.615;
   1:L PR[91] R[100]mm/sec CNT100;
   1:  PR[91,1] = PR[90,1] + 26.652;
   1:  PR[91,2] = PR[90,2] + 11.391;
   1:L PR[91] R[100]mm/sec CNT100;
   1:  PR[91,1] = PR[90,1] + 26.180;
   1:  PR[91,2] = PR[90,2] + 12.235;
   1:L PR[91] R[100]mm/sec CNT100;
   1:  PR[91,1] = PR[90,1] + 23.119;
   1:  PR[91,2] = PR[90,2] + 16.304;
   1:L PR[91] R[100]mm/sec CNT100;
   1:  PR[91,1] = PR[90,1] + 22.343;
   1:  PR[91,2] = PR[90,2] + 17.186;
   1:L PR[91] R[100]mm/sec CNT100;
   1:  PR[91,1] = PR[90,1] + 18.465;
   1:  PR[91,2] = PR[90,2] + 20.260;
   1:L PR[91] R[100]mm/sec CNT100;
   1:  PR[91,1] = PR[90,1] + 17.242;
   1:  PR[91,2] = PR[90,2] + 21.125;
   1:L PR[91] R[100]mm/sec CNT100;
   1:  PR[91,1] = PR[90,1] + 12.859;
   1:  PR[91,2] = PR[90,2] + 23.069;
   1:L PR[91] R[100]mm/sec CNT100;
   1:  PR[91,1] = PR[90,1] + 11.293;
   1:  PR[91,2] = PR[90,2] + 23.676;
   1:L PR[91] R[100]mm/sec CNT100;
   1:  PR[91,1] = PR[90,1] + 6.726;
   1:  PR[91,2] = PR[90,2] + 24.438;
   1:L PR[91] R[100]mm/sec CNT100;
   1:  PR[91,1] = PR[90,1] + 4.873;
   1:  PR[91,2] = PR[90,2] + 24.668;
   1:L PR[91] R[100]mm/sec CNT100;
   1:  PR[91,1] = PR[90,1] + 0.376;
   1:  PR[91,2] = PR[90,2] + 24.310;
   1:L PR[91] R[100]mm/sec CNT100;
   1:  PR[91] = PR[90];
   1:  PR[91,1] = PR[90,1] + -0.204;
   1:  PR[91,2] = PR[90,2] + 24.470;
   1:  PR[91,3] = PR[90,3] + 63.745;
   1:L PR[91] R[100]mm/sec CNT100;
   1:  PR[91,1] = PR[90,1] + -4.457;
   1:  PR[91,2] = PR[90,2] + 24.805;
   1:L PR[91] R[100]mm/sec CNT100;
   1:  PR[91,1] = PR[90,1] + -6.580;
   1:  PR[91,2] = PR[90,2] + 24.542;
   1:L PR[91] R[100]mm/sec CNT100;
   1:  PR[91,1] = PR[90,1] + -10.894;
   1:  PR[91,2] = PR[90,2] + 23.823;
   1:L PR[91] R[100]mm/sec CNT100;
   1:  PR[91,1] = PR[90,1] + -12.722;
   1:  PR[91,2] = PR[90,2] + 23.115;
   1:L PR[91] R[100]mm/sec CNT100;
   1:  PR[91,1] = PR[90,1] + -16.862;
   1:  PR[91,2] = PR[90,2] + 21.278;
   1:L PR[91] R[100]mm/sec CNT100;
   1:  PR[91,1] = PR[90,1] + -18.323;
   1:  PR[91,2] = PR[90,2] + 20.244;
   1:L PR[91] R[100]mm/sec CNT100;
   1:  PR[91,1] = PR[90,1] + -21.991;
   1:  PR[91,2] = PR[90,2] + 17.338;
   1:L PR[91] R[100]mm/sec CNT100;
   1:  PR[91,1] = PR[90,1] + -22.877;
   1:  PR[91,2] = PR[90,2] + 16.345;
   1:L PR[91] R[100]mm/sec CNT100;
   1:  PR[91,1] = PR[90,1] + -25.779;
   1:  PR[91,2] = PR[90,2] + 12.490;
   1:L PR[91] R[100]mm/sec CNT100;
   1:  PR[91,1] = PR[90,1] + -26.372;
   1:  PR[91,2] = PR[90,2] + 11.474;
   1:L PR[91] R[100]mm/sec CNT100;
   1:  PR[91,1] = PR[90,1] + -28.230;
   1:  PR[91,2] = PR[90,2] + 6.951;
   1:L PR[91] R[100]mm/sec CNT100;
   1:  PR[91,1] = PR[90,1] + -28.611;
   1:  PR[91,2] = PR[90,2] + 5.820;
   1:L PR[91] R[100]mm/sec CNT100;
   1:  PR[91,1] = PR[90,1] + -29.249;
   1:  PR[91,2] = PR[90,2] + 0.916;
   1:L PR[91] R[100]mm/sec CNT100;
   1:  PR[91,1] = PR[90,1] + -29.383;
   1:  PR[91,2] = PR[90,2] + -0.298;
   1:L PR[91] R[100]mm/sec CNT100;
   1:  PR[91,1] = PR[90,1] + -28.750;
   1:  PR[91,2] = PR[90,2] + -5.154;
   1:L PR[91] R[100]mm/sec CNT100;
   1:  PR[91,1] = PR[90,1] + -28.621;
   1:  PR[91,2] = PR[90,2] + -6.395;
   1:L PR[91] R[100]mm/sec CNT100;
   1:  PR[91,1] = PR[90,1] + -28.282;
   1:  PR[91,2] = PR[90,2] + -7.461;
   1:L PR[91] R[100]mm/sec CNT100;
   1:  PR[91,1] = PR[90,1] + -26.423;
   1:  PR[91,2] = PR[90,2] + -11.981;
   1:L PR[91] R[100]mm/sec CNT100;
   1:  PR[91,1] = PR[90,1] + -25.827;
   1:  PR[91,2] = PR[90,2] + -13.047;
   1:L PR[91] R[100]mm/sec CNT100;
   1:  PR[91,1] = PR[90,1] + -22.930;
   1:  PR[91,2] = PR[90,2] + -16.890;
   1:L PR[91] R[100]mm/sec CNT100;
   1:  PR[91,1] = PR[90,1] + -21.977;
   1:  PR[91,2] = PR[90,2] + -17.975;
   1:L PR[91] R[100]mm/sec CNT100;
   1:  PR[91,1] = PR[90,1] + -17.540;
   1:  PR[91,2] = PR[90,2] + -21.491;
   1:L PR[91] R[100]mm/sec CNT100;
   1:  PR[91,1] = PR[90,1] + -16.829;
   1:  PR[91,2] = PR[90,2] + -21.924;
   1:L PR[91] R[100]mm/sec CNT100;
   1:  PR[91,1] = PR[90,1] + -12.653;
   1:  PR[91,2] = PR[90,2] + -23.771;
   1:L PR[91] R[100]mm/sec CNT100;
   1:  PR[91,1] = PR[90,1] + -10.817;
   1:  PR[91,2] = PR[90,2] + -24.465;
   1:L PR[91] R[100]mm/sec CNT100;
   1:  PR[91,1] = PR[90,1] + -6.526;
   1:  PR[91,2] = PR[90,2] + -25.175;
   1:L PR[91] R[100]mm/sec CNT100;
   1:  PR[91,1] = PR[90,1] + -4.390;
   1:  PR[91,2] = PR[90,2] + -25.427;
   1:L PR[91] R[100]mm/sec CNT100;
   1:  PR[91,1] = PR[90,1] + -0.206;
   1:  PR[91,2] = PR[90,2] + -25.088;
   1:L PR[91] R[100]mm/sec CNT100;
   1:  PR[91,1] = PR[90,1] + 0.363;
   1:L PR[91] R[100]mm/sec CNT100;
   1:  PR[91,1] = PR[90,1] + 4.590;
   1:  PR[91,2] = PR[90,2] + -25.430;
   1:L PR[91] R[100]mm/sec CNT100;
   1:  PR[91,1] = PR[90,1] + 5.642;
   1:  PR[91,2] = PR[90,2] + -25.367;
   1:L PR[91] R[100]mm/sec CNT100;
   1:  PR[91,1] = PR[90,1] + 10.090;
   1:  PR[91,2] = PR[90,2] + -24.630;
   1:L PR[91] R[100]mm/sec CNT100;
   1:  PR[91,1] = PR[90,1] + 11.039;
   1:  PR[91,2] = PR[90,2] + -24.450;
   1:L PR[91] R[100]mm/sec CNT100;
   1:  PR[91,1] = PR[90,1] + 12.871;
   1:  PR[91,2] = PR[90,2] + -23.738;
   1:L PR[91] R[100]mm/sec CNT100;
   1:  PR[91,1] = PR[90,1] + 17.003;
   1:  PR[91,2] = PR[90,2] + -21.911;
   1:L PR[91] R[100]mm/sec CNT100;
   1:  PR[91,1] = PR[90,1] + 18.466;
   1:  PR[91,2] = PR[90,2] + -20.876;
   1:L PR[91] R[100]mm/sec CNT100;
   1:  PR[91,1] = PR[90,1] + 22.139;
   1:  PR[91,2] = PR[90,2] + -17.971;
   1:L PR[91] R[100]mm/sec CNT100;
   1:  PR[91,1] = PR[90,1] + 23.025;
   1:  PR[91,2] = PR[90,2] + -16.978;
   1:L PR[91] R[100]mm/sec CNT100;
   1:  PR[91,1] = PR[90,1] + 25.932;
   1:  PR[91,2] = PR[90,2] + -13.120;
   1:L PR[91] R[100]mm/sec CNT100;
   1:  PR[91,1] = PR[90,1] + 26.524;
   1:  PR[91,2] = PR[90,2] + -12.103;
   1:L PR[91] R[100]mm/sec CNT100;
   1:  PR[91,1] = PR[90,1] + 28.386;
   1:  PR[91,2] = PR[90,2] + -7.583;
   1:L PR[91] R[100]mm/sec CNT100;
   1:  PR[91,1] = PR[90,1] + 28.766;
   1:  PR[91,2] = PR[90,2] + -6.453;
   1:L PR[91] R[100]mm/sec CNT100;
   1:  PR[91,1] = PR[90,1] + 29.406;
   1:  PR[91,2] = PR[90,2] + -1.540;
   1:L PR[91] R[100]mm/sec CNT100;
   1:  PR[91,1] = PR[90,1] + 29.540;
   1:  PR[91,2] = PR[90,2] + -0.326;
   1:L PR[91] R[100]mm/sec CNT100;
   1:  PR[91,1] = PR[90,1] + 28.908;
   1:  PR[91,2] = PR[90,2] + 4.529;
   1:L PR[91] R[100]mm/sec CNT100;
   1:  PR[91,1] = PR[90,1] + 28.779;
   1:  PR[91,2] = PR[90,2] + 5.770;
   1:L PR[91] R[100]mm/sec CNT100;
   1:  PR[91,1] = PR[90,1] + 28.440;
   1:  PR[91,2] = PR[90,2] + 6.836;
   1:L PR[91] R[100]mm/sec CNT100;
   1:  PR[91,1] = PR[90,1] + 26.585;
   1:  PR[91,2] = PR[90,2] + 11.347;
   1:L PR[91] R[100]mm/sec CNT100;
   1:  PR[91,1] = PR[90,1] + 25.989;
   1:  PR[91,2] = PR[90,2] + 12.413;
   1:L PR[91] R[100]mm/sec CNT100;
   1:  PR[91,1] = PR[90,1] + 23.097;
   1:  PR[91,2] = PR[90,2] + 16.256;
   1:L PR[91] R[100]mm/sec CNT100;
   1:  PR[91,1] = PR[90,1] + 22.145;
   1:  PR[91,2] = PR[90,2] + 17.340;
   1:L PR[91] R[100]mm/sec CNT100;
   1:  PR[91,1] = PR[90,1] + 18.481;
   1:  PR[91,2] = PR[90,2] + 20.244;
   1:L PR[91] R[100]mm/sec CNT100;
   1:  PR[91,1] = PR[90,1] + 17.020;
   1:  PR[91,2] = PR[90,2] + 21.278;
   1:L PR[91] R[100]mm/sec CNT100;
   1:  PR[91,1] = PR[90,1] + 12.880;
   1:  PR[91,2] = PR[90,2] + 23.114;
   1:L PR[91] R[100]mm/sec CNT100;
   1:  PR[91,1] = PR[90,1] + 11.052;
   1:  PR[91,2] = PR[90,2] + 23.823;
   1:L PR[91] R[100]mm/sec CNT100;
   1:  PR[91,1] = PR[90,1] + 6.737;
   1:  PR[91,2] = PR[90,2] + 24.542;
   1:L PR[91] R[100]mm/sec CNT100;
   1:  PR[91,1] = PR[90,1] + 4.614;
   1:  PR[91,2] = PR[90,2] + 24.805;
   1:L PR[91] R[100]mm/sec CNT100;
   1:  PR[91,1] = PR[90,1] + 0.361;
   1:  PR[91,2] = PR[90,2] + 24.470;
   1:L PR[91] R[100]mm/sec CNT100;
   1:  PR[91] = PR[90];
   1:  PR[91,1] = PR[90,1] + -0.191;
   1:  PR[91,2] = PR[90,2] + 24.629;
   1:  PR[91,3] = PR[90,3] + 64.355;
   1:L PR[91] R[100]mm/sec CNT100;
   1:  PR[91,1] = PR[90,1] + -4.199;
   1:  PR[91,2] = PR[90,2] + 24.943;
   1:L PR[91] R[100]mm/sec CNT100;
   1:  PR[91,1] = PR[90,1] + -6.592;
   1:  PR[91,2] = PR[90,2] + 24.646;
   1:L PR[91] R[100]mm/sec CNT100;
   1:  PR[91,1] = PR[90,1] + -10.653;
   1:  PR[91,2] = PR[90,2] + 23.969;
   1:L PR[91] R[100]mm/sec CNT100;
   1:  PR[91,1] = PR[90,1] + -12.743;
   1:  PR[91,2] = PR[90,2] + 23.159;
   1:L PR[91] R[100]mm/sec CNT100;
   1:  PR[91,1] = PR[90,1] + -16.640;
   1:  PR[91,2] = PR[90,2] + 21.430;
   1:L PR[91] R[100]mm/sec CNT100;
   1:  PR[91,1] = PR[90,1] + -18.339;
   1:  PR[91,2] = PR[90,2] + 20.228;
   1:L PR[91] R[100]mm/sec CNT100;
   1:  PR[91,1] = PR[90,1] + -21.793;
   1:  PR[91,2] = PR[90,2] + 17.492;
   1:L PR[91] R[100]mm/sec CNT100;
   1:  PR[91,1] = PR[90,1] + -22.845;
   1:  PR[91,2] = PR[90,2] + 16.312;
   1:L PR[91] R[100]mm/sec CNT100;
   1:  PR[91,1] = PR[90,1] + -25.577;
   1:  PR[91,2] = PR[90,2] + 12.684;
   1:L PR[91] R[100]mm/sec CNT100;
   1:  PR[91,1] = PR[90,1] + -26.294;
   1:  PR[91,2] = PR[90,2] + 11.454;
   1:L PR[91] R[100]mm/sec CNT100;
   1:  PR[91,1] = PR[90,1] + -28.042;
   1:  PR[91,2] = PR[90,2] + 7.198;
   1:L PR[91] R[100]mm/sec CNT100;
   1:  PR[91,1] = PR[90,1] + -28.509;
   1:  PR[91,2] = PR[90,2] + 5.814;
   1:L PR[91] R[100]mm/sec CNT100;
   1:  PR[91,1] = PR[90,1] + -29.109;
   1:  PR[91,2] = PR[90,2] + 1.200;
   1:L PR[91] R[100]mm/sec CNT100;
   1:  PR[91,1] = PR[90,1] + -29.275;
   1:  PR[91,2] = PR[90,2] + -0.298;
   1:L PR[91] R[100]mm/sec CNT100;
   1:  PR[91,1] = PR[90,1] + -28.679;
   1:  PR[91,2] = PR[90,2] + -4.865;
   1:L PR[91] R[100]mm/sec CNT100;
   1:  PR[91,1] = PR[90,1] + -28.522;
   1:  PR[91,2] = PR[90,2] + -6.371;
   1:L PR[91] R[100]mm/sec CNT100;
   1:  PR[91,1] = PR[90,1] + -28.105;
   1:  PR[91,2] = PR[90,2] + -7.682;
   1:L PR[91] R[100]mm/sec CNT100;
   1:  PR[91,1] = PR[90,1] + -26.357;
   1:  PR[91,2] = PR[90,2] + -11.936;
   1:L PR[91] R[100]mm/sec CNT100;
   1:  PR[91,1] = PR[90,1] + -25.636;
   1:  PR[91,2] = PR[90,2] + -13.225;
   1:L PR[91] R[100]mm/sec CNT100;
   1:  PR[91,1] = PR[90,1] + -22.910;
   1:  PR[91,2] = PR[90,2] + -16.842;
   1:L PR[91] R[100]mm/sec CNT100;
   1:  PR[91,1] = PR[90,1] + -21.779;
   1:  PR[91,2] = PR[90,2] + -18.129;
   1:L PR[91] R[100]mm/sec CNT100;
   1:  PR[91,1] = PR[90,1] + -17.438;
   1:  PR[91,2] = PR[90,2] + -21.570;
   1:L PR[91] R[100]mm/sec CNT100;
   1:  PR[91,1] = PR[90,1] + -16.598;
   1:  PR[91,2] = PR[90,2] + -22.080;
   1:L PR[91] R[100]mm/sec CNT100;
   1:  PR[91,1] = PR[90,1] + -12.667;
   1:  PR[91,2] = PR[90,2] + -23.820;
   1:L PR[91] R[100]mm/sec CNT100;
   1:  PR[91,1] = PR[90,1] + -10.568;
   1:  PR[91,2] = PR[90,2] + -24.613;
   1:L PR[91] R[100]mm/sec CNT100;
   1:  PR[91,1] = PR[90,1] + -6.535;
   1:  PR[91,2] = PR[90,2] + -25.280;
   1:L PR[91] R[100]mm/sec CNT100;
   1:  PR[91,1] = PR[90,1] + -4.127;
   1:  PR[91,2] = PR[90,2] + -25.564;
   1:L PR[91] R[100]mm/sec CNT100;
   1:  PR[91,1] = PR[90,1] + -0.191;
   1:  PR[91,2] = PR[90,2] + -25.250;
   1:L PR[91] R[100]mm/sec CNT100;
   1:  PR[91,1] = PR[90,1] + 0.348;
   1:L PR[91] R[100]mm/sec CNT100;
   1:  PR[91,1] = PR[90,1] + 4.326;
   1:  PR[91,2] = PR[90,2] + -25.567;
   1:L PR[91] R[100]mm/sec CNT100;
   1:  PR[91,1] = PR[90,1] + 5.525;
   1:  PR[91,2] = PR[90,2] + -25.496;
   1:L PR[91] R[100]mm/sec CNT100;
   1:  PR[91,1] = PR[90,1] + 9.709;
   1:  PR[91,2] = PR[90,2] + -24.802;
   1:L PR[91] R[100]mm/sec CNT100;
   1:  PR[91,1] = PR[90,1] + 10.801;
   1:  PR[91,2] = PR[90,2] + -24.595;
   1:L PR[91] R[100]mm/sec CNT100;
   1:  PR[91,1] = PR[90,1] + 12.894;
   1:  PR[91,2] = PR[90,2] + -23.782;
   1:L PR[91] R[100]mm/sec CNT100;
   1:  PR[91,1] = PR[90,1] + 16.781;
   1:  PR[91,2] = PR[90,2] + -22.063;
   1:L PR[91] R[100]mm/sec CNT100;
   1:  PR[91,1] = PR[90,1] + 18.483;
   1:  PR[91,2] = PR[90,2] + -20.860;
   1:L PR[91] R[100]mm/sec CNT100;
   1:  PR[91,1] = PR[90,1] + 21.941;
   1:  PR[91,2] = PR[90,2] + -18.124;
   1:L PR[91] R[100]mm/sec CNT100;
   1:  PR[91,1] = PR[90,1] + 22.994;
   1:  PR[91,2] = PR[90,2] + -16.944;
   1:L PR[91] R[100]mm/sec CNT100;
   1:  PR[91,1] = PR[90,1] + 25.729;
   1:  PR[91,2] = PR[90,2] + -13.313;
   1:L PR[91] R[100]mm/sec CNT100;
   1:  PR[91,1] = PR[90,1] + 26.447;
   1:  PR[91,2] = PR[90,2] + -12.083;
   1:L PR[91] R[100]mm/sec CNT100;
   1:  PR[91,1] = PR[90,1] + 28.198;
   1:  PR[91,2] = PR[90,2] + -7.829;
   1:L PR[91] R[100]mm/sec CNT100;
   1:  PR[91,1] = PR[90,1] + 28.664;
   1:  PR[91,2] = PR[90,2] + -6.446;
   1:L PR[91] R[100]mm/sec CNT100;
   1:  PR[91,1] = PR[90,1] + 29.266;
   1:  PR[91,2] = PR[90,2] + -1.824;
   1:L PR[91] R[100]mm/sec CNT100;
   1:  PR[91,1] = PR[90,1] + 29.432;
   1:  PR[91,2] = PR[90,2] + -0.326;
   1:L PR[91] R[100]mm/sec CNT100;
   1:  PR[91,1] = PR[90,1] + 28.837;
   1:  PR[91,2] = PR[90,2] + 4.241;
   1:L PR[91] R[100]mm/sec CNT100;
   1:  PR[91,1] = PR[90,1] + 28.680;
   1:  PR[91,2] = PR[90,2] + 5.747;
   1:L PR[91] R[100]mm/sec CNT100;
   1:  PR[91,1] = PR[90,1] + 28.264;
   1:  PR[91,2] = PR[90,2] + 7.057;
   1:L PR[91] R[100]mm/sec CNT100;
   1:  PR[91,1] = PR[90,1] + 26.518;
   1:  PR[91,2] = PR[90,2] + 11.302;
   1:L PR[91] R[100]mm/sec CNT100;
   1:  PR[91,1] = PR[90,1] + 25.798;
   1:  PR[91,2] = PR[90,2] + 12.591;
   1:L PR[91] R[100]mm/sec CNT100;
   1:  PR[91,1] = PR[90,1] + 23.076;
   1:  PR[91,2] = PR[90,2] + 16.208;
   1:L PR[91] R[100]mm/sec CNT100;
   1:  PR[91,1] = PR[90,1] + 21.946;
   1:  PR[91,2] = PR[90,2] + 17.494;
   1:L PR[91] R[100]mm/sec CNT100;
   1:  PR[91,1] = PR[90,1] + 18.496;
   1:  PR[91,2] = PR[90,2] + 20.228;
   1:L PR[91] R[100]mm/sec CNT100;
   1:  PR[91,1] = PR[90,1] + 16.798;
   1:  PR[91,2] = PR[90,2] + 21.430;
   1:L PR[91] R[100]mm/sec CNT100;
   1:  PR[91,1] = PR[90,1] + 12.901;
   1:  PR[91,2] = PR[90,2] + 23.159;
   1:L PR[91] R[100]mm/sec CNT100;
   1:  PR[91,1] = PR[90,1] + 10.810;
   1:  PR[91,2] = PR[90,2] + 23.969;
   1:L PR[91] R[100]mm/sec CNT100;
   1:  PR[91,1] = PR[90,1] + 6.749;
   1:  PR[91,2] = PR[90,2] + 24.646;
   1:L PR[91] R[100]mm/sec CNT100;
   1:  PR[91,1] = PR[90,1] + 4.356;
   1:  PR[91,2] = PR[90,2] + 24.943;
   1:L PR[91] R[100]mm/sec CNT100;
   1:  PR[91,1] = PR[90,1] + 0.348;
   1:  PR[91,2] = PR[90,2] + 24.629;
   1:L PR[91] R[100]mm/sec CNT100;
   1:  PR[91] = PR[90];
   1:  PR[91,1] = PR[90,1] + -0.177;
   1:  PR[91,2] = PR[90,2] + 24.787;
   1:  PR[91,3] = PR[90,3] + 64.965;
   1:L PR[91] R[100]mm/sec CNT100;
   1:  PR[91,1] = PR[90,1] + -3.941;
   1:  PR[91,2] = PR[90,2] + 25.080;
   1:L PR[91] R[100]mm/sec CNT100;
   1:  PR[91,1] = PR[90,1] + -6.604;
   1:  PR[91,2] = PR[90,2] + 24.750;
   1:L PR[91] R[100]mm/sec CNT100;
   1:  PR[91,1] = PR[90,1] + -10.411;
   1:  PR[91,2] = PR[90,2] + 24.116;
   1:L PR[91] R[100]mm/sec CNT100;
   1:  PR[91,1] = PR[90,1] + -12.764;
   1:  PR[91,2] = PR[90,2] + 23.204;
   1:L PR[91] R[100]mm/sec CNT100;
   1:  PR[91,1] = PR[90,1] + -16.418;
   1:  PR[91,2] = PR[90,2] + 21.583;
   1:L PR[91] R[100]mm/sec CNT100;
   1:  PR[91,1] = PR[90,1] + -18.354;
   1:  PR[91,2] = PR[90,2] + 20.212;
   1:L PR[91] R[100]mm/sec CNT100;
   1:  PR[91,1] = PR[90,1] + -21.594;
   1:  PR[91,2] = PR[90,2] + 17.646;
   1:L PR[91] R[100]mm/sec CNT100;
   1:  PR[91,1] = PR[90,1] + -22.813;
   1:  PR[91,2] = PR[90,2] + 16.280;
   1:L PR[91] R[100]mm/sec CNT100;
   1:  PR[91,1] = PR[90,1] + -25.374;
   1:  PR[91,2] = PR[90,2] + 12.877;
   1:L PR[91] R[100]mm/sec CNT100;
   1:  PR[91,1] = PR[90,1] + -26.216;
   1:  PR[91,2] = PR[90,2] + 11.434;
   1:L PR[91] R[100]mm/sec CNT100;
   1:  PR[91,1] = PR[90,1] + -27.854;
   1:  PR[91,2] = PR[90,2] + 7.444;
   1:L PR[91] R[100]mm/sec CNT100;
   1:  PR[91,1] = PR[90,1] + -28.407;
   1:  PR[91,2] = PR[90,2] + 5.807;
   1:L PR[91] R[100]mm/sec CNT100;
   1:  PR[91,1] = PR[90,1] + -28.969;
   1:  PR[91,2] = PR[90,2] + 1.484;
   1:L PR[91] R[100]mm/sec CNT100;
   1:  PR[91,1] = PR[90,1] + -29.167;
   1:  PR[91,2] = PR[90,2] + -0.298;
   1:L PR[91] R[100]mm/sec CNT100;
   1:  PR[91,1] = PR[90,1] + -28.608;
   1:  PR[91,2] = PR[90,2] + -4.577;
   1:L PR[91] R[100]mm/sec CNT100;
   1:  PR[91,1] = PR[90,1] + -28.424;
   1:  PR[91,2] = PR[90,2] + -6.348;
   1:L PR[91] R[100]mm/sec CNT100;
   1:  PR[91,1] = PR[90,1] + -27.929;
   1:  PR[91,2] = PR[90,2] + -7.903;
   1:L PR[91] R[100]mm/sec CNT100;
   1:  PR[91,1] = PR[90,1] + -26.290;
   1:  PR[91,2] = PR[90,2] + -11.890;
   1:L PR[91] R[100]mm/sec CNT100;
   1:  PR[91,1] = PR[90,1] + -25.445;
   1:  PR[91,2] = PR[90,2] + -13.402;
   1:L PR[91] R[100]mm/sec CNT100;
   1:  PR[91,1] = PR[90,1] + -22.889;
   1:  PR[91,2] = PR[90,2] + -16.793;
   1:L PR[91] R[100]mm/sec CNT100;
   1:  PR[91,1] = PR[90,1] + -21.580;
   1:  PR[91,2] = PR[90,2] + -18.282;
   1:L PR[91] R[100]mm/sec CNT100;
   1:  PR[91,1] = PR[90,1] + -17.335;
   1:  PR[91,2] = PR[90,2] + -21.649;
   1:L PR[91] R[100]mm/sec CNT100;
   1:  PR[91,1] = PR[90,1] + -16.368;
   1:  PR[91,2] = PR[90,2] + -22.237;
   1:L PR[91] R[100]mm/sec CNT100;
   1:  PR[91,1] = PR[90,1] + -12.682;
   1:  PR[91,2] = PR[90,2] + -23.868;
   1:L PR[91] R[100]mm/sec CNT100;
   1:  PR[91,1] = PR[90,1] + -10.319;
   1:  PR[91,2] = PR[90,2] + -24.761;
   1:L PR[91] R[100]mm/sec CNT100;
   1:  PR[91,1] = PR[90,1] + -6.544;
   1:  PR[91,2] = PR[90,2] + -25.385;
   1:L PR[91] R[100]mm/sec CNT100;
   1:  PR[91,1] = PR[90,1] + -3.864;
   1:  PR[91,2] = PR[90,2] + -25.701;
   1:L PR[91] R[100]mm/sec CNT100;
   1:  PR[91,1] = PR[90,1] + -0.176;
   1:  PR[91,2] = PR[90,2] + -25.413;
   1:L PR[91] R[100]mm/sec CNT100;
   1:  PR[91,1] = PR[90,1] + 0.333;
   1:L PR[91] R[100]mm/sec CNT100;
   1:  PR[91,1] = PR[90,1] + 4.063;
   1:  PR[91,2] = PR[90,2] + -25.705;
   1:L PR[91] R[100]mm/sec CNT100;
   1:  PR[91,1] = PR[90,1] + 5.407;
   1:  PR[91,2] = PR[90,2] + -25.624;
   1:L PR[91] R[100]mm/sec CNT100;
   1:  PR[91,1] = PR[90,1] + 9.327;
   1:  PR[91,2] = PR[90,2] + -24.974;
   1:L PR[91] R[100]mm/sec CNT100;
   1:  PR[91,1] = PR[90,1] + 10.564;
   1:  PR[91,2] = PR[90,2] + -24.740;
   1:L PR[91] R[100]mm/sec CNT100;
   1:  PR[91,1] = PR[90,1] + 12.918;
   1:  PR[91,2] = PR[90,2] + -23.825;
   1:L PR[91] R[100]mm/sec CNT100;
   1:  PR[91,1] = PR[90,1] + 16.560;
   1:  PR[91,2] = PR[90,2] + -22.215;
   1:L PR[91] R[100]mm/sec CNT100;
   1:  PR[91,1] = PR[90,1] + 18.499;
   1:  PR[91,2] = PR[90,2] + -20.843;
   1:L PR[91] R[100]mm/sec CNT100;
   1:  PR[91,1] = PR[90,1] + 21.743;
   1:  PR[91,2] = PR[90,2] + -18.278;
   1:L PR[91] R[100]mm/sec CNT100;
   1:  PR[91,1] = PR[90,1] + 22.962;
   1:  PR[91,2] = PR[90,2] + -16.911;
   1:L PR[91] R[100]mm/sec CNT100;
   1:  PR[91,1] = PR[90,1] + 25.527;
   1:  PR[91,2] = PR[90,2] + -13.506;
   1:L PR[91] R[100]mm/sec CNT100;
   1:  PR[91,1] = PR[90,1] + 26.369;
   1:  PR[91,2] = PR[90,2] + -12.062;
   1:L PR[91] R[100]mm/sec CNT100;
   1:  PR[91,1] = PR[90,1] + 28.011;
   1:  PR[91,2] = PR[90,2] + -8.075;
   1:L PR[91] R[100]mm/sec CNT100;
   1:  PR[91,1] = PR[90,1] + 28.562;
   1:  PR[91,2] = PR[90,2] + -6.438;
   1:L PR[91] R[100]mm/sec CNT100;
   1:  PR[91,1] = PR[90,1] + 29.126;
   1:  PR[91,2] = PR[90,2] + -2.108;
   1:L PR[91] R[100]mm/sec CNT100;
   1:  PR[91,1] = PR[90,1] + 29.323;
   1:  PR[91,2] = PR[90,2] + -0.326;
   1:L PR[91] R[100]mm/sec CNT100;
   1:  PR[91,1] = PR[90,1] + 28.766;
   1:  PR[91,2] = PR[90,2] + 3.953;
   1:L PR[91] R[100]mm/sec CNT100;
   1:  PR[91,1] = PR[90,1] + 28.582;
   1:  PR[91,2] = PR[90,2] + 5.723;
   1:L PR[91] R[100]mm/sec CNT100;
   1:  PR[91,1] = PR[90,1] + 28.087;
   1:  PR[91,2] = PR[90,2] + 7.278;
   1:L PR[91] R[100]mm/sec CNT100;
   1:  PR[91,1] = PR[90,1] + 26.451;
   1:  PR[91,2] = PR[90,2] + 11.257;
   1:L PR[91] R[100]mm/sec CNT100;
   1:  PR[91,1] = PR[90,1] + 25.606;
   1:  PR[91,2] = PR[90,2] + 12.769;
   1:L PR[91] R[100]mm/sec CNT100;
   1:  PR[91,1] = PR[90,1] + 23.054;
   1:  PR[91,2] = PR[90,2] + 16.161;
   1:L PR[91] R[100]mm/sec CNT100;
   1:  PR[91,1] = PR[90,1] + 21.747;
   1:  PR[91,2] = PR[90,2] + 17.649;
   1:L PR[91] R[100]mm/sec CNT100;
   1:  PR[91,1] = PR[90,1] + 18.512;
   1:  PR[91,2] = PR[90,2] + 20.212;
   1:L PR[91] R[100]mm/sec CNT100;
   1:  PR[91,1] = PR[90,1] + 16.576;
   1:  PR[91,2] = PR[90,2] + 21.583;
   1:L PR[91] R[100]mm/sec CNT100;
   1:  PR[91,1] = PR[90,1] + 12.922;
   1:  PR[91,2] = PR[90,2] + 23.203;
   1:L PR[91] R[100]mm/sec CNT100;
   1:  PR[91,1] = PR[90,1] + 10.568;
   1:  PR[91,2] = PR[90,2] + 24.115;
   1:L PR[91] R[100]mm/sec CNT100;
   1:  PR[91,1] = PR[90,1] + 6.761;
   1:  PR[91,2] = PR[90,2] + 24.751;
   1:L PR[91] R[100]mm/sec CNT100;
   1:  PR[91,1] = PR[90,1] + 4.098;
   1:  PR[91,2] = PR[90,2] + 25.080;
   1:L PR[91] R[100]mm/sec CNT100;
   1:  PR[91,1] = PR[90,1] + 0.334;
   1:  PR[91,2] = PR[90,2] + 24.787;
   1:L PR[91] R[100]mm/sec CNT100;
   1:  PR[91] = PR[90];
   1:  PR[91,1] = PR[90,1] + -0.164;
   1:  PR[91,2] = PR[90,2] + 24.945;
   1:  PR[91,3] = PR[90,3] + 65.575;
   1:L PR[91] R[100]mm/sec CNT100;
   1:  PR[91,1] = PR[90,1] + -3.682;
   1:  PR[91,2] = PR[90,2] + 25.218;
   1:L PR[91] R[100]mm/sec CNT100;
   1:  PR[91,1] = PR[90,1] + -6.616;
   1:  PR[91,2] = PR[90,2] + 24.855;
   1:L PR[91] R[100]mm/sec CNT100;
   1:  PR[91,1] = PR[90,1] + -10.169;
   1:  PR[91,2] = PR[90,2] + 24.262;
   1:L PR[91] R[100]mm/sec CNT100;
   1:  PR[91,1] = PR[90,1] + -12.785;
   1:  PR[91,2] = PR[90,2] + 23.249;
   1:L PR[91] R[100]mm/sec CNT100;
   1:  PR[91,1] = PR[90,1] + -16.196;
   1:  PR[91,2] = PR[90,2] + 21.735;
   1:L PR[91] R[100]mm/sec CNT100;
   1:  PR[91,1] = PR[90,1] + -18.370;
   1:  PR[91,2] = PR[90,2] + 20.196;
   1:L PR[91] R[100]mm/sec CNT100;
   1:  PR[91,1] = PR[90,1] + -21.395;
   1:  PR[91,2] = PR[90,2] + 17.800;
   1:L PR[91] R[100]mm/sec CNT100;
   1:  PR[91,1] = PR[90,1] + -22.780;
   1:  PR[91,2] = PR[90,2] + 16.247;
   1:L PR[91] R[100]mm/sec CNT100;
   1:  PR[91,1] = PR[90,1] + -25.172;
   1:  PR[91,2] = PR[90,2] + 13.070;
   1:L PR[91] R[100]mm/sec CNT100;
   1:  PR[91,1] = PR[90,1] + -26.138;
   1:  PR[91,2] = PR[90,2] + 11.414;
   1:L PR[91] R[100]mm/sec CNT100;
   1:  PR[91,1] = PR[90,1] + -27.667;
   1:  PR[91,2] = PR[90,2] + 7.691;
   1:L PR[91] R[100]mm/sec CNT100;
   1:  PR[91,1] = PR[90,1] + -28.305;
   1:  PR[91,2] = PR[90,2] + 5.800;
   1:L PR[91] R[100]mm/sec CNT100;
   1:  PR[91,1] = PR[90,1] + -28.829;
   1:  PR[91,2] = PR[90,2] + 1.768;
   1:L PR[91] R[100]mm/sec CNT100;
   1:  PR[91,1] = PR[90,1] + -29.058;
   1:  PR[91,2] = PR[90,2] + -0.298;
   1:L PR[91] R[100]mm/sec CNT100;
   1:  PR[91,1] = PR[90,1] + -28.538;
   1:  PR[91,2] = PR[90,2] + -4.288;
   1:L PR[91] R[100]mm/sec CNT100;
   1:  PR[91,1] = PR[90,1] + -28.325;
   1:  PR[91,2] = PR[90,2] + -6.325;
   1:L PR[91] R[100]mm/sec CNT100;
   1:  PR[91,1] = PR[90,1] + -27.753;
   1:  PR[91,2] = PR[90,2] + -8.125;
   1:L PR[91] R[100]mm/sec CNT100;
   1:  PR[91,1] = PR[90,1] + -26.223;
   1:  PR[91,2] = PR[90,2] + -11.845;
   1:L PR[91] R[100]mm/sec CNT100;
   1:  PR[91,1] = PR[90,1] + -25.254;
   1:  PR[91,2] = PR[90,2] + -13.579;
   1:L PR[91] R[100]mm/sec CNT100;
   1:  PR[91,1] = PR[90,1] + -22.868;
   1:  PR[91,2] = PR[90,2] + -16.745;
   1:L PR[91] R[100]mm/sec CNT100;
   1:  PR[91,1] = PR[90,1] + -21.382;
   1:  PR[91,2] = PR[90,2] + -18.436;
   1:L PR[91] R[100]mm/sec CNT100;
   1:  PR[91,1] = PR[90,1] + -17.232;
   1:  PR[91,2] = PR[90,2] + -21.727;
   1:L PR[91] R[100]mm/sec CNT100;
   1:  PR[91,1] = PR[90,1] + -16.137;
   1:  PR[91,2] = PR[90,2] + -22.394;
   1:L PR[91] R[100]mm/sec CNT100;
   1:  PR[91,1] = PR[90,1] + -12.697;
   1:  PR[91,2] = PR[90,2] + -23.916;
   1:L PR[91] R[100]mm/sec CNT100;
   1:  PR[91,1] = PR[90,1] + -10.071;
   1:  PR[91,2] = PR[90,2] + -24.909;
   1:L PR[91] R[100]mm/sec CNT100;
   1:  PR[91,1] = PR[90,1] + -6.553;
   1:  PR[91,2] = PR[90,2] + -25.490;
   1:L PR[91] R[100]mm/sec CNT100;
   1:  PR[91,1] = PR[90,1] + -3.601;
   1:  PR[91,2] = PR[90,2] + -25.838;
   1:L PR[91] R[100]mm/sec CNT100;
   1:  PR[91,1] = PR[90,1] + -0.163;
   1:  PR[91,2] = PR[90,2] + -25.571;
   1:L PR[91] R[100]mm/sec CNT100;
   1:  PR[91,1] = PR[90,1] + 0.319;
   1:L PR[91] R[100]mm/sec CNT100;
   1:  PR[91,1] = PR[90,1] + 3.801;
   1:  PR[91,2] = PR[90,2] + -25.842;
   1:L PR[91] R[100]mm/sec CNT100;
   1:  PR[91,1] = PR[90,1] + 5.289;
   1:  PR[91,2] = PR[90,2] + -25.753;
   1:L PR[91] R[100]mm/sec CNT100;
   1:  PR[91,1] = PR[90,1] + 8.946;
   1:  PR[91,2] = PR[90,2] + -25.146;
   1:L PR[91] R[100]mm/sec CNT100;
   1:  PR[91,1] = PR[90,1] + 10.326;
   1:  PR[91,2] = PR[90,2] + -24.885;
   1:L PR[91] R[100]mm/sec CNT100;
   1:  PR[91,1] = PR[90,1] + 12.941;
   1:  PR[91,2] = PR[90,2] + -23.869;
   1:L PR[91] R[100]mm/sec CNT100;
   1:  PR[91,1] = PR[90,1] + 16.338;
   1:  PR[91,2] = PR[90,2] + -22.367;
   1:L PR[91] R[100]mm/sec CNT100;
   1:  PR[91,1] = PR[90,1] + 18.516;
   1:  PR[91,2] = PR[90,2] + -20.827;
   1:L PR[91] R[100]mm/sec CNT100;
   1:  PR[91,1] = PR[90,1] + 21.545;
   1:  PR[91,2] = PR[90,2] + -18.431;
   1:L PR[91] R[100]mm/sec CNT100;
   1:  PR[91,1] = PR[90,1] + 22.930;
   1:  PR[91,2] = PR[90,2] + -16.878;
   1:L PR[91] R[100]mm/sec CNT100;
   1:  PR[91,1] = PR[90,1] + 25.325;
   1:  PR[91,2] = PR[90,2] + -13.699;
   1:L PR[91] R[100]mm/sec CNT100;
   1:  PR[91,1] = PR[90,1] + 26.291;
   1:  PR[91,2] = PR[90,2] + -12.042;
   1:L PR[91] R[100]mm/sec CNT100;
   1:  PR[91,1] = PR[90,1] + 27.823;
   1:  PR[91,2] = PR[90,2] + -8.321;
   1:L PR[91] R[100]mm/sec CNT100;
   1:  PR[91,1] = PR[90,1] + 28.460;
   1:  PR[91,2] = PR[90,2] + -6.431;
   1:L PR[91] R[100]mm/sec CNT100;
   1:  PR[91,1] = PR[90,1] + 28.986;
   1:  PR[91,2] = PR[90,2] + -2.392;
   1:L PR[91] R[100]mm/sec CNT100;
   1:  PR[91,1] = PR[90,1] + 29.215;
   1:  PR[91,2] = PR[90,2] + -0.326;
   1:L PR[91] R[100]mm/sec CNT100;
   1:  PR[91,1] = PR[90,1] + 28.695;
   1:  PR[91,2] = PR[90,2] + 3.664;
   1:L PR[91] R[100]mm/sec CNT100;
   1:  PR[91,1] = PR[90,1] + 28.483;
   1:  PR[91,2] = PR[90,2] + 5.700;
   1:L PR[91] R[100]mm/sec CNT100;
   1:  PR[91,1] = PR[90,1] + 27.911;
   1:  PR[91,2] = PR[90,2] + 7.500;
   1:L PR[91] R[100]mm/sec CNT100;
   1:  PR[91,1] = PR[90,1] + 26.384;
   1:  PR[91,2] = PR[90,2] + 11.212;
   1:L PR[91] R[100]mm/sec CNT100;
   1:  PR[91,1] = PR[90,1] + 25.415;
   1:  PR[91,2] = PR[90,2] + 12.947;
   1:L PR[91] R[100]mm/sec CNT100;
   1:  PR[91,1] = PR[90,1] + 23.033;
   1:  PR[91,2] = PR[90,2] + 16.113;
   1:L PR[91] R[100]mm/sec CNT100;
   1:  PR[91,1] = PR[90,1] + 21.548;
   1:  PR[91,2] = PR[90,2] + 17.803;
   1:L PR[91] R[100]mm/sec CNT100;
   1:  PR[91,1] = PR[90,1] + 18.527;
   1:  PR[91,2] = PR[90,2] + 20.196;
   1:L PR[91] R[100]mm/sec CNT100;
   1:  PR[91,1] = PR[90,1] + 16.354;
   1:  PR[91,2] = PR[90,2] + 21.735;
   1:L PR[91] R[100]mm/sec CNT100;
   1:  PR[91,1] = PR[90,1] + 12.942;
   1:  PR[91,2] = PR[90,2] + 23.248;
   1:L PR[91] R[100]mm/sec CNT100;
   1:  PR[91,1] = PR[90,1] + 10.326;
   1:  PR[91,2] = PR[90,2] + 24.262;
   1:L PR[91] R[100]mm/sec CNT100;
   1:  PR[91,1] = PR[90,1] + 6.773;
   1:  PR[91,2] = PR[90,2] + 24.855;
   1:L PR[91] R[100]mm/sec CNT100;
   1:  PR[91,1] = PR[90,1] + 3.839;
   1:  PR[91,2] = PR[90,2] + 25.218;
   1:L PR[91] R[100]mm/sec CNT100;
   1:  PR[91,1] = PR[90,1] + 0.321;
   1:  PR[91,2] = PR[90,2] + 24.945;
   1:L PR[91] R[100]mm/sec CNT100;
   1:  PR[91] = PR[90];
   1:  PR[91,1] = PR[90,1] + -0.150;
   1:  PR[91,2] = PR[90,2] + 25.103;
   1:  PR[91,3] = PR[90,3] + 66.185;
   1:L PR[91] R[100]mm/sec CNT100;
   1:  PR[91,1] = PR[90,1] + -3.424;
   1:  PR[91,2] = PR[90,2] + 25.356;
   1:L PR[91] R[100]mm/sec CNT100;
   1:  PR[91,1] = PR[90,1] + -6.628;
   1:  PR[91,2] = PR[90,2] + 24.959;
   1:L PR[91] R[100]mm/sec CNT100;
   1:  PR[91,1] = PR[90,1] + -9.928;
   1:  PR[91,2] = PR[90,2] + 24.409;
   1:L PR[91] R[100]mm/sec CNT100;
   1:  PR[91,1] = PR[90,1] + -12.806;
   1:  PR[91,2] = PR[90,2] + 23.293;
   1:L PR[91] R[100]mm/sec CNT100;
   1:  PR[91,1] = PR[90,1] + -15.974;
   1:  PR[91,2] = PR[90,2] + 21.888;
   1:L PR[91] R[100]mm/sec CNT100;
   1:  PR[91,1] = PR[90,1] + -18.385;
   1:  PR[91,2] = PR[90,2] + 20.180;
   1:L PR[91] R[100]mm/sec CNT100;
   1:  PR[91,1] = PR[90,1] + -21.196;
   1:  PR[91,2] = PR[90,2] + 17.954;
   1:L PR[91] R[100]mm/sec CNT100;
   1:  PR[91,1] = PR[90,1] + -22.748;
   1:  PR[91,2] = PR[90,2] + 16.214;
   1:L PR[91] R[100]mm/sec CNT100;
   1:  PR[91,1] = PR[90,1] + -24.969;
   1:  PR[91,2] = PR[90,2] + 13.264;
   1:L PR[91] R[100]mm/sec CNT100;
   1:  PR[91,1] = PR[90,1] + -26.060;
   1:  PR[91,2] = PR[90,2] + 11.394;
   1:L PR[91] R[100]mm/sec CNT100;
   1:  PR[91,1] = PR[90,1] + -27.479;
   1:  PR[91,2] = PR[90,2] + 7.938;
   1:L PR[91] R[100]mm/sec CNT100;
   1:  PR[91,1] = PR[90,1] + -28.203;
   1:  PR[91,2] = PR[90,2] + 5.794;
   1:L PR[91] R[100]mm/sec CNT100;
   1:  PR[91,1] = PR[90,1] + -28.689;
   1:  PR[91,2] = PR[90,2] + 2.052;
   1:L PR[91] R[100]mm/sec CNT100;
   1:  PR[91,1] = PR[90,1] + -28.950;
   1:  PR[91,2] = PR[90,2] + -0.298;
   1:L PR[91] R[100]mm/sec CNT100;
   1:  PR[91,1] = PR[90,1] + -28.467;
   1:  PR[91,2] = PR[90,2] + -4.000;
   1:L PR[91] R[100]mm/sec CNT100;
   1:  PR[91,1] = PR[90,1] + -28.227;
   1:  PR[91,2] = PR[90,2] + -6.301;
   1:L PR[91] R[100]mm/sec CNT100;
   1:  PR[91,1] = PR[90,1] + -27.577;
   1:  PR[91,2] = PR[90,2] + -8.346;
   1:L PR[91] R[100]mm/sec CNT100;
   1:  PR[91,1] = PR[90,1] + -26.157;
   1:  PR[91,2] = PR[90,2] + -11.800;
   1:L PR[91] R[100]mm/sec CNT100;
   1:  PR[91,1] = PR[90,1] + -25.063;
   1:  PR[91,2] = PR[90,2] + -13.757;
   1:L PR[91] R[100]mm/sec CNT100;
   1:  PR[91,1] = PR[90,1] + -22.847;
   1:  PR[91,2] = PR[90,2] + -16.697;
   1:L PR[91] R[100]mm/sec CNT100;
   1:  PR[91,1] = PR[90,1] + -21.183;
   1:  PR[91,2] = PR[90,2] + -18.590;
   1:L PR[91] R[100]mm/sec CNT100;
   1:  PR[91,1] = PR[90,1] + -17.129;
   1:  PR[91,2] = PR[90,2] + -21.806;
   1:L PR[91] R[100]mm/sec CNT100;
   1:  PR[91,1] = PR[90,1] + -15.906;
   1:  PR[91,2] = PR[90,2] + -22.551;
   1:L PR[91] R[100]mm/sec CNT100;
   1:  PR[91,1] = PR[90,1] + -12.712;
   1:  PR[91,2] = PR[90,2] + -23.964;
   1:L PR[91] R[100]mm/sec CNT100;
   1:  PR[91,1] = PR[90,1] + -9.822;
   1:  PR[91,2] = PR[90,2] + -25.057;
   1:L PR[91] R[100]mm/sec CNT100;
   1:  PR[91,1] = PR[90,1] + -6.562;
   1:  PR[91,2] = PR[90,2] + -25.596;
   1:L PR[91] R[100]mm/sec CNT100;
   1:  PR[91,1] = PR[90,1] + -3.339;
   1:  PR[91,2] = PR[90,2] + -25.976;
   1:L PR[91] R[100]mm/sec CNT100;
   1:  PR[91,1] = PR[90,1] + -0.150;
   1:  PR[91,2] = PR[90,2] + -25.728;
   1:L PR[91] R[100]mm/sec CNT100;
   1:  PR[91,1] = PR[90,1] + 0.307;
   1:L PR[91] R[100]mm/sec CNT100;
   1:  PR[91,1] = PR[90,1] + 3.539;
   1:  PR[91,2] = PR[90,2] + -25.979;
   1:L PR[91] R[100]mm/sec CNT100;
   1:  PR[91,1] = PR[90,1] + 5.171;
   1:  PR[91,2] = PR[90,2] + -25.881;
   1:L PR[91] R[100]mm/sec CNT100;
   1:  PR[91,1] = PR[90,1] + 8.565;
   1:  PR[91,2] = PR[90,2] + -25.318;
   1:L PR[91] R[100]mm/sec CNT100;
   1:  PR[91,1] = PR[90,1] + 10.088;
   1:  PR[91,2] = PR[90,2] + -25.031;
   1:L PR[91] R[100]mm/sec CNT100;
   1:  PR[91,1] = PR[90,1] + 12.965;
   1:  PR[91,2] = PR[90,2] + -23.912;
   1:L PR[91] R[100]mm/sec CNT100;
   1:  PR[91,1] = PR[90,1] + 16.116;
   1:  PR[91,2] = PR[90,2] + -22.519;
   1:L PR[91] R[100]mm/sec CNT100;
   1:  PR[91,1] = PR[90,1] + 18.532;
   1:  PR[91,2] = PR[90,2] + -20.811;
   1:L PR[91] R[100]mm/sec CNT100;
   1:  PR[91,1] = PR[90,1] + 21.346;
   1:  PR[91,2] = PR[90,2] + -18.585;
   1:L PR[91] R[100]mm/sec CNT100;
   1:  PR[91,1] = PR[90,1] + 22.898;
   1:  PR[91,2] = PR[90,2] + -16.845;
   1:L PR[91] R[100]mm/sec CNT100;
   1:  PR[91,1] = PR[90,1] + 25.123;
   1:  PR[91,2] = PR[90,2] + -13.891;
   1:L PR[91] R[100]mm/sec CNT100;
   1:  PR[91,1] = PR[90,1] + 26.214;
   1:  PR[91,2] = PR[90,2] + -12.021;
   1:L PR[91] R[100]mm/sec CNT100;
   1:  PR[91,1] = PR[90,1] + 27.636;
   1:  PR[91,2] = PR[90,2] + -8.567;
   1:L PR[91] R[100]mm/sec CNT100;
   1:  PR[91,1] = PR[90,1] + 28.358;
   1:  PR[91,2] = PR[90,2] + -6.424;
   1:L PR[91] R[100]mm/sec CNT100;
   1:  PR[91,1] = PR[90,1] + 28.846;
   1:  PR[91,2] = PR[90,2] + -2.676;
   1:L PR[91] R[100]mm/sec CNT100;
   1:  PR[91,1] = PR[90,1] + 29.107;
   1:  PR[91,2] = PR[90,2] + -0.326;
   1:L PR[91] R[100]mm/sec CNT100;
   1:  PR[91,1] = PR[90,1] + 28.625;
   1:  PR[91,2] = PR[90,2] + 3.376;
   1:L PR[91] R[100]mm/sec CNT100;
   1:  PR[91,1] = PR[90,1] + 28.385;
   1:  PR[91,2] = PR[90,2] + 5.677;
   1:L PR[91] R[100]mm/sec CNT100;
   1:  PR[91,1] = PR[90,1] + 27.735;
   1:  PR[91,2] = PR[90,2] + 7.721;
   1:L PR[91] R[100]mm/sec CNT100;
   1:  PR[91,1] = PR[90,1] + 26.317;
   1:  PR[91,2] = PR[90,2] + 11.167;
   1:L PR[91] R[100]mm/sec CNT100;
   1:  PR[91,1] = PR[90,1] + 25.224;
   1:  PR[91,2] = PR[90,2] + 13.125;
   1:L PR[91] R[100]mm/sec CNT100;
   1:  PR[91,1] = PR[90,1] + 23.011;
   1:  PR[91,2] = PR[90,2] + 16.065;
   1:L PR[91] R[100]mm/sec CNT100;
   1:  PR[91,1] = PR[90,1] + 21.349;
   1:  PR[91,2] = PR[90,2] + 17.957;
   1:L PR[91] R[100]mm/sec CNT100;
   1:  PR[91,1] = PR[90,1] + 18.543;
   1:  PR[91,2] = PR[90,2] + 20.180;
   1:L PR[91] R[100]mm/sec CNT100;
   1:  PR[91,1] = PR[90,1] + 16.131;
   1:  PR[91,2] = PR[90,2] + 21.888;
   1:L PR[91] R[100]mm/sec CNT100;
   1:  PR[91,1] = PR[90,1] + 12.963;
   1:  PR[91,2] = PR[90,2] + 23.293;
   1:L PR[91] R[100]mm/sec CNT100;
   1:  PR[91,1] = PR[90,1] + 10.085;
   1:  PR[91,2] = PR[90,2] + 24.408;
   1:L PR[91] R[100]mm/sec CNT100;
   1:  PR[91,1] = PR[90,1] + 6.785;
   1:  PR[91,2] = PR[90,2] + 24.959;
   1:L PR[91] R[100]mm/sec CNT100;
   1:  PR[91,1] = PR[90,1] + 3.581;
   1:  PR[91,2] = PR[90,2] + 25.356;
   1:L PR[91] R[100]mm/sec CNT100;
   1:  PR[91,1] = PR[90,1] + 0.307;
   1:  PR[91,2] = PR[90,2] + 25.103;
   1:L PR[91] R[100]mm/sec CNT100;
   1:  PR[91] = PR[90];
   1:  PR[91,1] = PR[90,1] + -0.137;
   1:  PR[91,2] = PR[90,2] + 25.261;
   1:  PR[91,3] = PR[90,3] + 66.795;
   1:L PR[91] R[100]mm/sec CNT100;
   1:  PR[91,1] = PR[90,1] + -3.166;
   1:  PR[91,2] = PR[90,2] + 25.493;
   1:L PR[91] R[100]mm/sec CNT100;
   1:  PR[91,1] = PR[90,1] + -6.639;
   1:  PR[91,2] = PR[90,2] + 25.063;
   1:L PR[91] R[100]mm/sec CNT100;
   1:  PR[91,1] = PR[90,1] + -9.686;
   1:  PR[91,2] = PR[90,2] + 24.555;
   1:L PR[91] R[100]mm/sec CNT100;
   1:  PR[91,1] = PR[90,1] + -12.827;
   1:  PR[91,2] = PR[90,2] + 23.338;
   1:L PR[91] R[100]mm/sec CNT100;
   1:  PR[91,1] = PR[90,1] + -15.752;
   1:  PR[91,2] = PR[90,2] + 22.040;
   1:L PR[91] R[100]mm/sec CNT100;
   1:  PR[91,1] = PR[90,1] + -18.401;
   1:  PR[91,2] = PR[90,2] + 20.165;
   1:L PR[91] R[100]mm/sec CNT100;
   1:  PR[91,1] = PR[90,1] + -20.997;
   1:  PR[91,2] = PR[90,2] + 18.108;
   1:L PR[91] R[100]mm/sec CNT100;
   1:  PR[91,1] = PR[90,1] + -22.716;
   1:  PR[91,2] = PR[90,2] + 16.182;
   1:L PR[91] R[100]mm/sec CNT100;
   1:  PR[91,1] = PR[90,1] + -24.767;
   1:  PR[91,2] = PR[90,2] + 13.457;
   1:L PR[91] R[100]mm/sec CNT100;
   1:  PR[91,1] = PR[90,1] + -25.982;
   1:  PR[91,2] = PR[90,2] + 11.374;
   1:L PR[91] R[100]mm/sec CNT100;
   1:  PR[91,1] = PR[90,1] + -27.292;
   1:  PR[91,2] = PR[90,2] + 8.184;
   1:L PR[91] R[100]mm/sec CNT100;
   1:  PR[91,1] = PR[90,1] + -28.100;
   1:  PR[91,2] = PR[90,2] + 5.787;
   1:L PR[91] R[100]mm/sec CNT100;
   1:  PR[91,1] = PR[90,1] + -28.549;
   1:  PR[91,2] = PR[90,2] + 2.336;
   1:L PR[91] R[100]mm/sec CNT100;
   1:  PR[91,1] = PR[90,1] + -28.841;
   1:  PR[91,2] = PR[90,2] + -0.298;
   1:L PR[91] R[100]mm/sec CNT100;
   1:  PR[91,1] = PR[90,1] + -28.396;
   1:  PR[91,2] = PR[90,2] + -3.712;
   1:L PR[91] R[100]mm/sec CNT100;
   1:  PR[91,1] = PR[90,1] + -28.128;
   1:  PR[91,2] = PR[90,2] + -6.278;
   1:L PR[91] R[100]mm/sec CNT100;
   1:  PR[91,1] = PR[90,1] + -27.400;
   1:  PR[91,2] = PR[90,2] + -8.567;
   1:L PR[91] R[100]mm/sec CNT100;
   1:  PR[91,1] = PR[90,1] + -26.090;
   1:  PR[91,2] = PR[90,2] + -11.754;
   1:L PR[91] R[100]mm/sec CNT100;
   1:  PR[91,1] = PR[90,1] + -24.872;
   1:  PR[91,2] = PR[90,2] + -13.934;
   1:L PR[91] R[100]mm/sec CNT100;
   1:  PR[91,1] = PR[90,1] + -22.826;
   1:  PR[91,2] = PR[90,2] + -16.648;
   1:L PR[91] R[100]mm/sec CNT100;
   1:  PR[91,1] = PR[90,1] + -20.985;
   1:  PR[91,2] = PR[90,2] + -18.743;
   1:L PR[91] R[100]mm/sec CNT100;
   1:  PR[91,1] = PR[90,1] + -17.027;
   1:  PR[91,2] = PR[90,2] + -21.885;
   1:L PR[91] R[100]mm/sec CNT100;
   1:  PR[91,1] = PR[90,1] + -15.676;
   1:  PR[91,2] = PR[90,2] + -22.708;
   1:L PR[91] R[100]mm/sec CNT100;
   1:  PR[91,1] = PR[90,1] + -12.727;
   1:  PR[91,2] = PR[90,2] + -24.012;
   1:L PR[91] R[100]mm/sec CNT100;
   1:  PR[91,1] = PR[90,1] + -9.573;
   1:  PR[91,2] = PR[90,2] + -25.204;
   1:L PR[91] R[100]mm/sec CNT100;
   1:  PR[91,1] = PR[90,1] + -6.572;
   1:  PR[91,2] = PR[90,2] + -25.701;
   1:L PR[91] R[100]mm/sec CNT100;
   1:  PR[91,1] = PR[90,1] + -3.077;
   1:  PR[91,2] = PR[90,2] + -26.113;
   1:L PR[91] R[100]mm/sec CNT100;
   1:  PR[91,1] = PR[90,1] + -0.137;
   1:  PR[91,2] = PR[90,2] + -25.884;
   1:L PR[91] R[100]mm/sec CNT100;
   1:  PR[91,1] = PR[90,1] + 0.294;
   1:L PR[91] R[100]mm/sec CNT100;
   1:  PR[91,1] = PR[90,1] + 3.277;
   1:  PR[91,2] = PR[90,2] + -26.116;
   1:L PR[91] R[100]mm/sec CNT100;
   1:  PR[91,1] = PR[90,1] + 5.053;
   1:  PR[91,2] = PR[90,2] + -26.010;
   1:L PR[91] R[100]mm/sec CNT100;
   1:  PR[91,1] = PR[90,1] + 8.183;
   1:  PR[91,2] = PR[90,2] + -25.491;
   1:L PR[91] R[100]mm/sec CNT100;
   1:  PR[91,1] = PR[90,1] + 9.851;
   1:  PR[91,2] = PR[90,2] + -25.176;
   1:L PR[91] R[100]mm/sec CNT100;
   1:  PR[91,1] = PR[90,1] + 12.988;
   1:  PR[91,2] = PR[90,2] + -23.956;
   1:L PR[91] R[100]mm/sec CNT100;
   1:  PR[91,1] = PR[90,1] + 15.895;
   1:  PR[91,2] = PR[90,2] + -22.671;
   1:L PR[91] R[100]mm/sec CNT100;
   1:  PR[91,1] = PR[90,1] + 18.548;
   1:  PR[91,2] = PR[90,2] + -20.794;
   1:L PR[91] R[100]mm/sec CNT100;
   1:  PR[91,1] = PR[90,1] + 21.148;
   1:  PR[91,2] = PR[90,2] + -18.738;
   1:L PR[91] R[100]mm/sec CNT100;
   1:  PR[91,1] = PR[90,1] + 22.867;
   1:  PR[91,2] = PR[90,2] + -16.812;
   1:L PR[91] R[100]mm/sec CNT100;
   1:  PR[91,1] = PR[90,1] + 24.921;
   1:  PR[91,2] = PR[90,2] + -14.084;
   1:L PR[91] R[100]mm/sec CNT100;
   1:  PR[91,1] = PR[90,1] + 26.136;
   1:  PR[91,2] = PR[90,2] + -12.001;
   1:L PR[91] R[100]mm/sec CNT100;
   1:  PR[91,1] = PR[90,1] + 27.448;
   1:  PR[91,2] = PR[90,2] + -8.813;
   1:L PR[91] R[100]mm/sec CNT100;
   1:  PR[91,1] = PR[90,1] + 28.256;
   1:  PR[91,2] = PR[90,2] + -6.417;
   1:L PR[91] R[100]mm/sec CNT100;
   1:  PR[91,1] = PR[90,1] + 28.706;
   1:  PR[91,2] = PR[90,2] + -2.960;
   1:L PR[91] R[100]mm/sec CNT100;
   1:  PR[91,1] = PR[90,1] + 28.998;
   1:  PR[91,2] = PR[90,2] + -0.326;
   1:L PR[91] R[100]mm/sec CNT100;
   1:  PR[91,1] = PR[90,1] + 28.554;
   1:  PR[91,2] = PR[90,2] + 3.088;
   1:L PR[91] R[100]mm/sec CNT100;
   1:  PR[91,1] = PR[90,1] + 28.286;
   1:  PR[91,2] = PR[90,2] + 5.653;
   1:L PR[91] R[100]mm/sec CNT100;
   1:  PR[91,1] = PR[90,1] + 27.558;
   1:  PR[91,2] = PR[90,2] + 7.942;
   1:L PR[91] R[100]mm/sec CNT100;
   1:  PR[91,1] = PR[90,1] + 26.251;
   1:  PR[91,2] = PR[90,2] + 11.122;
   1:L PR[91] R[100]mm/sec CNT100;
   1:  PR[91,1] = PR[90,1] + 25.032;
   1:  PR[91,2] = PR[90,2] + 13.302;
   1:L PR[91] R[100]mm/sec CNT100;
   1:  PR[91,1] = PR[90,1] + 22.990;
   1:  PR[91,2] = PR[90,2] + 16.017;
   1:L PR[91] R[100]mm/sec CNT100;
   1:  PR[91,1] = PR[90,1] + 21.150;
   1:  PR[91,2] = PR[90,2] + 18.111;
   1:L PR[91] R[100]mm/sec CNT100;
   1:  PR[91,1] = PR[90,1] + 18.558;
   1:  PR[91,2] = PR[90,2] + 20.164;
   1:L PR[91] R[100]mm/sec CNT100;
   1:  PR[91,1] = PR[90,1] + 15.909;
   1:  PR[91,2] = PR[90,2] + 22.040;
   1:L PR[91] R[100]mm/sec CNT100;
   1:  PR[91,1] = PR[90,1] + 12.984;
   1:  PR[91,2] = PR[90,2] + 23.338;
   1:L PR[91] R[100]mm/sec CNT100;
   1:  PR[91,1] = PR[90,1] + 9.843;
   1:  PR[91,2] = PR[90,2] + 24.555;
   1:L PR[91] R[100]mm/sec CNT100;
   1:  PR[91,1] = PR[90,1] + 6.796;
   1:  PR[91,2] = PR[90,2] + 25.063;
   1:L PR[91] R[100]mm/sec CNT100;
   1:  PR[91,1] = PR[90,1] + 3.322;
   1:  PR[91,2] = PR[90,2] + 25.493;
   1:L PR[91] R[100]mm/sec CNT100;
   1:  PR[91,1] = PR[90,1] + 0.293;
   1:  PR[91,2] = PR[90,2] + 25.261;
   1:L PR[91] R[100]mm/sec CNT100;
   1:  PR[91] = PR[90];
   1:  PR[91,1] = PR[90,1] + -0.123;
   1:  PR[91,2] = PR[90,2] + 25.419;
   1:  PR[91,3] = PR[90,3] + 67.405;
   1:L PR[91] R[100]mm/sec CNT100;
   1:  PR[91,1] = PR[90,1] + -2.907;
   1:  PR[91,2] = PR[90,2] + 25.631;
   1:L PR[91] R[100]mm/sec CNT100;
   1:  PR[91,1] = PR[90,1] + -6.651;
   1:  PR[91,2] = PR[90,2] + 25.167;
   1:L PR[91] R[100]mm/sec CNT100;
   1:  PR[91,1] = PR[90,1] + -9.444;
   1:  PR[91,2] = PR[90,2] + 24.701;
   1:L PR[91] R[100]mm/sec CNT100;
   1:  PR[91,1] = PR[90,1] + -12.848;
   1:  PR[91,2] = PR[90,2] + 23.383;
   1:L PR[91] R[100]mm/sec CNT100;
   1:  PR[91,1] = PR[90,1] + -15.530;
   1:  PR[91,2] = PR[90,2] + 22.193;
   1:L PR[91] R[100]mm/sec CNT100;
   1:  PR[91,1] = PR[90,1] + -18.416;
   1:  PR[91,2] = PR[90,2] + 20.149;
   1:L PR[91] R[100]mm/sec CNT100;
   1:  PR[91,1] = PR[90,1] + -20.798;
   1:  PR[91,2] = PR[90,2] + 18.262;
   1:L PR[91] R[100]mm/sec CNT100;
   1:  PR[91,1] = PR[90,1] + -22.683;
   1:  PR[91,2] = PR[90,2] + 16.149;
   1:L PR[91] R[100]mm/sec CNT100;
   1:  PR[91,1] = PR[90,1] + -24.564;
   1:  PR[91,2] = PR[90,2] + 13.650;
   1:L PR[91] R[100]mm/sec CNT100;
   1:  PR[91,1] = PR[90,1] + -25.904;
   1:  PR[91,2] = PR[90,2] + 11.354;
   1:L PR[91] R[100]mm/sec CNT100;
   1:  PR[91,1] = PR[90,1] + -27.104;
   1:  PR[91,2] = PR[90,2] + 8.431;
   1:L PR[91] R[100]mm/sec CNT100;
   1:  PR[91,1] = PR[90,1] + -27.998;
   1:  PR[91,2] = PR[90,2] + 5.780;
   1:L PR[91] R[100]mm/sec CNT100;
   1:  PR[91,1] = PR[90,1] + -28.409;
   1:  PR[91,2] = PR[90,2] + 2.620;
   1:L PR[91] R[100]mm/sec CNT100;
   1:  PR[91,1] = PR[90,1] + -28.733;
   1:  PR[91,2] = PR[90,2] + -0.298;
   1:L PR[91] R[100]mm/sec CNT100;
   1:  PR[91,1] = PR[90,1] + -28.325;
   1:  PR[91,2] = PR[90,2] + -3.423;
   1:L PR[91] R[100]mm/sec CNT100;
   1:  PR[91,1] = PR[90,1] + -28.030;
   1:  PR[91,2] = PR[90,2] + -6.255;
   1:L PR[91] R[100]mm/sec CNT100;
   1:  PR[91,1] = PR[90,1] + -27.224;
   1:  PR[91,2] = PR[90,2] + -8.788;
   1:L PR[91] R[100]mm/sec CNT100;
   1:  PR[91,1] = PR[90,1] + -26.023;
   1:  PR[91,2] = PR[90,2] + -11.709;
   1:L PR[91] R[100]mm/sec CNT100;
   1:  PR[91,1] = PR[90,1] + -24.681;
   1:  PR[91,2] = PR[90,2] + -14.111;
   1:L PR[91] R[100]mm/sec CNT100;
   1:  PR[91,1] = PR[90,1] + -22.805;
   1:  PR[91,2] = PR[90,2] + -16.600;
   1:L PR[91] R[100]mm/sec CNT100;
   1:  PR[91,1] = PR[90,1] + -20.787;
   1:  PR[91,2] = PR[90,2] + -18.897;
   1:L PR[91] R[100]mm/sec CNT100;
   1:  PR[91,1] = PR[90,1] + -16.924;
   1:  PR[91,2] = PR[90,2] + -21.964;
   1:L PR[91] R[100]mm/sec CNT100;
   1:  PR[91,1] = PR[90,1] + -15.445;
   1:  PR[91,2] = PR[90,2] + -22.864;
   1:L PR[91] R[100]mm/sec CNT100;
   1:  PR[91,1] = PR[90,1] + -12.741;
   1:  PR[91,2] = PR[90,2] + -24.060;
   1:L PR[91] R[100]mm/sec CNT100;
   1:  PR[91,1] = PR[90,1] + -9.325;
   1:  PR[91,2] = PR[90,2] + -25.352;
   1:L PR[91] R[100]mm/sec CNT100;
   1:  PR[91,1] = PR[90,1] + -6.581;
   1:  PR[91,2] = PR[90,2] + -25.806;
   1:L PR[91] R[100]mm/sec CNT100;
   1:  PR[91,1] = PR[90,1] + -2.815;
   1:  PR[91,2] = PR[90,2] + -26.250;
   1:L PR[91] R[100]mm/sec CNT100;
   1:  PR[91,1] = PR[90,1] + -0.125;
   1:  PR[91,2] = PR[90,2] + -26.041;
   1:L PR[91] R[100]mm/sec CNT100;
   1:  PR[91,1] = PR[90,1] + 0.281;
   1:L PR[91] R[100]mm/sec CNT100;
   1:  PR[91,1] = PR[90,1] + 3.014;
   1:  PR[91,2] = PR[90,2] + -26.253;
   1:L PR[91] R[100]mm/sec CNT100;
   1:  PR[91,1] = PR[90,1] + 4.935;
   1:  PR[91,2] = PR[90,2] + -26.138;
   1:L PR[91] R[100]mm/sec CNT100;
   1:  PR[91,1] = PR[90,1] + 7.802;
   1:  PR[91,2] = PR[90,2] + -25.663;
   1:L PR[91] R[100]mm/sec CNT100;
   1:  PR[91,1] = PR[90,1] + 9.613;
   1:  PR[91,2] = PR[90,2] + -25.321;
   1:L PR[91] R[100]mm/sec CNT100;
   1:  PR[91,1] = PR[90,1] + 13.012;
   1:  PR[91,2] = PR[90,2] + -24.000;
   1:L PR[91] R[100]mm/sec CNT100;
   1:  PR[91,1] = PR[90,1] + 15.673;
   1:  PR[91,2] = PR[90,2] + -22.823;
   1:L PR[91] R[100]mm/sec CNT100;
   1:  PR[91,1] = PR[90,1] + 18.565;
   1:  PR[91,2] = PR[90,2] + -20.778;
   1:L PR[91] R[100]mm/sec CNT100;
   1:  PR[91,1] = PR[90,1] + 20.950;
   1:  PR[91,2] = PR[90,2] + -18.891;
   1:L PR[91] R[100]mm/sec CNT100;
   1:  PR[91,1] = PR[90,1] + 22.835;
   1:  PR[91,2] = PR[90,2] + -16.778;
   1:L PR[91] R[100]mm/sec CNT100;
   1:  PR[91,1] = PR[90,1] + 24.719;
   1:  PR[91,2] = PR[90,2] + -14.277;
   1:L PR[91] R[100]mm/sec CNT100;
   1:  PR[91,1] = PR[90,1] + 26.058;
   1:  PR[91,2] = PR[90,2] + -11.981;
   1:L PR[91] R[100]mm/sec CNT100;
   1:  PR[91,1] = PR[90,1] + 27.261;
   1:  PR[91,2] = PR[90,2] + -9.059;
   1:L PR[91] R[100]mm/sec CNT100;
   1:  PR[91,1] = PR[90,1] + 28.154;
   1:  PR[91,2] = PR[90,2] + -6.409;
   1:L PR[91] R[100]mm/sec CNT100;
   1:  PR[91,1] = PR[90,1] + 28.566;
   1:  PR[91,2] = PR[90,2] + -3.244;
   1:L PR[91] R[100]mm/sec CNT100;
   1:  PR[91,1] = PR[90,1] + 28.890;
   1:  PR[91,2] = PR[90,2] + -0.326;
   1:L PR[91] R[100]mm/sec CNT100;
   1:  PR[91,1] = PR[90,1] + 28.483;
   1:  PR[91,2] = PR[90,2] + 2.799;
   1:L PR[91] R[100]mm/sec CNT100;
   1:  PR[91,1] = PR[90,1] + 28.188;
   1:  PR[91,2] = PR[90,2] + 5.630;
   1:L PR[91] R[100]mm/sec CNT100;
   1:  PR[91,1] = PR[90,1] + 27.382;
   1:  PR[91,2] = PR[90,2] + 8.163;
   1:L PR[91] R[100]mm/sec CNT100;
   1:  PR[91,1] = PR[90,1] + 26.184;
   1:  PR[91,2] = PR[90,2] + 11.077;
   1:L PR[91] R[100]mm/sec CNT100;
   1:  PR[91,1] = PR[90,1] + 24.841;
   1:  PR[91,2] = PR[90,2] + 13.480;
   1:L PR[91] R[100]mm/sec CNT100;
   1:  PR[91,1] = PR[90,1] + 22.969;
   1:  PR[91,2] = PR[90,2] + 15.969;
   1:L PR[91] R[100]mm/sec CNT100;
   1:  PR[91,1] = PR[90,1] + 20.951;
   1:  PR[91,2] = PR[90,2] + 18.265;
   1:L PR[91] R[100]mm/sec CNT100;
   1:  PR[91,1] = PR[90,1] + 18.574;
   1:  PR[91,2] = PR[90,2] + 20.148;
   1:L PR[91] R[100]mm/sec CNT100;
   1:  PR[91,1] = PR[90,1] + 15.687;
   1:  PR[91,2] = PR[90,2] + 22.193;
   1:L PR[91] R[100]mm/sec CNT100;
   1:  PR[91,1] = PR[90,1] + 13.005;
   1:  PR[91,2] = PR[90,2] + 23.382;
   1:L PR[91] R[100]mm/sec CNT100;
   1:  PR[91,1] = PR[90,1] + 9.601;
   1:  PR[91,2] = PR[90,2] + 24.701;
   1:L PR[91] R[100]mm/sec CNT100;
   1:  PR[91,1] = PR[90,1] + 6.808;
   1:  PR[91,2] = PR[90,2] + 25.167;
   1:L PR[91] R[100]mm/sec CNT100;
   1:  PR[91,1] = PR[90,1] + 3.064;
   1:  PR[91,2] = PR[90,2] + 25.631;
   1:L PR[91] R[100]mm/sec CNT100;
   1:  PR[91,1] = PR[90,1] + 0.279;
   1:  PR[91,2] = PR[90,2] + 25.419;
   1:L PR[91] R[100]mm/sec CNT100;
   1:  PR[91] = PR[90];
   1:  PR[91,1] = PR[90,1] + -0.109;
   1:  PR[91,2] = PR[90,2] + 25.578;
   1:  PR[91,3] = PR[90,3] + 68.015;
   1:L PR[91] R[100]mm/sec CNT100;
   1:  PR[91,1] = PR[90,1] + -2.649;
   1:  PR[91,2] = PR[90,2] + 25.769;
   1:L PR[91] R[100]mm/sec CNT100;
   1:  PR[91,1] = PR[90,1] + -6.663;
   1:  PR[91,2] = PR[90,2] + 25.271;
   1:L PR[91] R[100]mm/sec CNT100;
   1:  PR[91,1] = PR[90,1] + -9.203;
   1:  PR[91,2] = PR[90,2] + 24.848;
   1:L PR[91] R[100]mm/sec CNT100;
   1:  PR[91,1] = PR[90,1] + -12.869;
   1:  PR[91,2] = PR[90,2] + 23.427;
   1:L PR[91] R[100]mm/sec CNT100;
   1:  PR[91,1] = PR[90,1] + -15.307;
   1:  PR[91,2] = PR[90,2] + 22.345;
   1:L PR[91] R[100]mm/sec CNT100;
   1:  PR[91,1] = PR[90,1] + -18.432;
   1:  PR[91,2] = PR[90,2] + 20.133;
   1:L PR[91] R[100]mm/sec CNT100;
   1:  PR[91,1] = PR[90,1] + -20.599;
   1:  PR[91,2] = PR[90,2] + 18.416;
   1:L PR[91] R[100]mm/sec CNT100;
   1:  PR[91,1] = PR[90,1] + -22.651;
   1:  PR[91,2] = PR[90,2] + 16.116;
   1:L PR[91] R[100]mm/sec CNT100;
   1:  PR[91,1] = PR[90,1] + -24.362;
   1:  PR[91,2] = PR[90,2] + 13.844;
   1:L PR[91] R[100]mm/sec CNT100;
   1:  PR[91,1] = PR[90,1] + -25.826;
   1:  PR[91,2] = PR[90,2] + 11.334;
   1:L PR[91] R[100]mm/sec CNT100;
   1:  PR[91,1] = PR[90,1] + -26.917;
   1:  PR[91,2] = PR[90,2] + 8.678;
   1:L PR[91] R[100]mm/sec CNT100;
   1:  PR[91,1] = PR[90,1] + -27.896;
   1:  PR[91,2] = PR[90,2] + 5.773;
   1:L PR[91] R[100]mm/sec CNT100;
   1:  PR[91,1] = PR[90,1] + -28.270;
   1:  PR[91,2] = PR[90,2] + 2.904;
   1:L PR[91] R[100]mm/sec CNT100;
   1:  PR[91,1] = PR[90,1] + -28.624;
   1:  PR[91,2] = PR[90,2] + -0.298;
   1:L PR[91] R[100]mm/sec CNT100;
   1:  PR[91,1] = PR[90,1] + -28.254;
   1:  PR[91,2] = PR[90,2] + -3.135;
   1:L PR[91] R[100]mm/sec CNT100;
   1:  PR[91,1] = PR[90,1] + -27.932;
   1:  PR[91,2] = PR[90,2] + -6.231;
   1:L PR[91] R[100]mm/sec CNT100;
   1:  PR[91,1] = PR[90,1] + -27.048;
   1:  PR[91,2] = PR[90,2] + -9.010;
   1:L PR[91] R[100]mm/sec CNT100;
   1:  PR[91,1] = PR[90,1] + -25.957;
   1:  PR[91,2] = PR[90,2] + -11.663;
   1:L PR[91] R[100]mm/sec CNT100;
   1:  PR[91,1] = PR[90,1] + -24.490;
   1:  PR[91,2] = PR[90,2] + -14.289;
   1:L PR[91] R[100]mm/sec CNT100;
   1:  PR[91,1] = PR[90,1] + -22.784;
   1:  PR[91,2] = PR[90,2] + -16.551;
   1:L PR[91] R[100]mm/sec CNT100;
   1:  PR[91,1] = PR[90,1] + -20.588;
   1:  PR[91,2] = PR[90,2] + -19.050;
   1:L PR[91] R[100]mm/sec CNT100;
   1:  PR[91,1] = PR[90,1] + -16.821;
   1:  PR[91,2] = PR[90,2] + -22.043;
   1:L PR[91] R[100]mm/sec CNT100;
   1:  PR[91,1] = PR[90,1] + -15.214;
   1:  PR[91,2] = PR[90,2] + -23.021;
   1:L PR[91] R[100]mm/sec CNT100;
   1:  PR[91,1] = PR[90,1] + -12.756;
   1:  PR[91,2] = PR[90,2] + -24.109;
   1:L PR[91] R[100]mm/sec CNT100;
   1:  PR[91,1] = PR[90,1] + -9.076;
   1:  PR[91,2] = PR[90,2] + -25.500;
   1:L PR[91] R[100]mm/sec CNT100;
   1:  PR[91,1] = PR[90,1] + -6.590;
   1:  PR[91,2] = PR[90,2] + -25.911;
   1:L PR[91] R[100]mm/sec CNT100;
   1:  PR[91,1] = PR[90,1] + -2.553;
   1:  PR[91,2] = PR[90,2] + -26.387;
   1:L PR[91] R[100]mm/sec CNT100;
   1:  PR[91,1] = PR[90,1] + -0.112;
   1:  PR[91,2] = PR[90,2] + -26.197;
   1:L PR[91] R[100]mm/sec CNT100;
   1:  PR[91,1] = PR[90,1] + 0.269;
   1:L PR[91] R[100]mm/sec CNT100;
   1:  PR[91,1] = PR[90,1] + 2.752;
   1:  PR[91,2] = PR[90,2] + -26.390;
   1:L PR[91] R[100]mm/sec CNT100;
   1:  PR[91,1] = PR[90,1] + 4.818;
   1:  PR[91,2] = PR[90,2] + -26.267;
   1:L PR[91] R[100]mm/sec CNT100;
   1:  PR[91,1] = PR[90,1] + 7.421;
   1:  PR[91,2] = PR[90,2] + -25.835;
   1:L PR[91] R[100]mm/sec CNT100;
   1:  PR[91,1] = PR[90,1] + 9.376;
   1:  PR[91,2] = PR[90,2] + -25.466;
   1:L PR[91] R[100]mm/sec CNT100;
   1:  PR[91,1] = PR[90,1] + 13.035;
   1:  PR[91,2] = PR[90,2] + -24.043;
   1:L PR[91] R[100]mm/sec CNT100;
   1:  PR[91,1] = PR[90,1] + 15.451;
   1:  PR[91,2] = PR[90,2] + -22.975;
   1:L PR[91] R[100]mm/sec CNT100;
   1:  PR[91,1] = PR[90,1] + 18.581;
   1:  PR[91,2] = PR[90,2] + -20.762;
   1:L PR[91] R[100]mm/sec CNT100;
   1:  PR[91,1] = PR[90,1] + 20.751;
   1:  PR[91,2] = PR[90,2] + -19.045;
   1:L PR[91] R[100]mm/sec CNT100;
   1:  PR[91,1] = PR[90,1] + 22.803;
   1:  PR[91,2] = PR[90,2] + -16.745;
   1:L PR[91] R[100]mm/sec CNT100;
   1:  PR[91,1] = PR[90,1] + 24.517;
   1:  PR[91,2] = PR[90,2] + -14.470;
   1:L PR[91] R[100]mm/sec CNT100;
   1:  PR[91,1] = PR[90,1] + 25.981;
   1:  PR[91,2] = PR[90,2] + -11.960;
   1:L PR[91] R[100]mm/sec CNT100;
   1:  PR[91,1] = PR[90,1] + 27.074;
   1:  PR[91,2] = PR[90,2] + -9.305;
   1:L PR[91] R[100]mm/sec CNT100;
   1:  PR[91,1] = PR[90,1] + 28.052;
   1:  PR[91,2] = PR[90,2] + -6.402;
   1:L PR[91] R[100]mm/sec CNT100;
   1:  PR[91,1] = PR[90,1] + 28.426;
   1:  PR[91,2] = PR[90,2] + -3.528;
   1:L PR[91] R[100]mm/sec CNT100;
   1:  PR[91,1] = PR[90,1] + 28.781;
   1:  PR[91,2] = PR[90,2] + -0.326;
   1:L PR[91] R[100]mm/sec CNT100;
   1:  PR[91,1] = PR[90,1] + 28.412;
   1:  PR[91,2] = PR[90,2] + 2.511;
   1:L PR[91] R[100]mm/sec CNT100;
   1:  PR[91,1] = PR[90,1] + 28.089;
   1:  PR[91,2] = PR[90,2] + 5.607;
   1:L PR[91] R[100]mm/sec CNT100;
   1:  PR[91,1] = PR[90,1] + 27.206;
   1:  PR[91,2] = PR[90,2] + 8.384;
   1:L PR[91] R[100]mm/sec CNT100;
   1:  PR[91,1] = PR[90,1] + 26.117;
   1:  PR[91,2] = PR[90,2] + 11.033;
   1:L PR[91] R[100]mm/sec CNT100;
   1:  PR[91,1] = PR[90,1] + 24.650;
   1:  PR[91,2] = PR[90,2] + 13.658;
   1:L PR[91] R[100]mm/sec CNT100;
   1:  PR[91,1] = PR[90,1] + 22.947;
   1:  PR[91,2] = PR[90,2] + 15.921;
   1:L PR[91] R[100]mm/sec CNT100;
   1:  PR[91,1] = PR[90,1] + 20.753;
   1:  PR[91,2] = PR[90,2] + 18.419;
   1:L PR[91] R[100]mm/sec CNT100;
   1:  PR[91,1] = PR[90,1] + 18.590;
   1:  PR[91,2] = PR[90,2] + 20.133;
   1:L PR[91] R[100]mm/sec CNT100;
   1:  PR[91,1] = PR[90,1] + 15.465;
   1:  PR[91,2] = PR[90,2] + 22.345;
   1:L PR[91] R[100]mm/sec CNT100;
   1:  PR[91,1] = PR[90,1] + 13.026;
   1:  PR[91,2] = PR[90,2] + 23.427;
   1:L PR[91] R[100]mm/sec CNT100;
   1:  PR[91,1] = PR[90,1] + 9.359;
   1:  PR[91,2] = PR[90,2] + 24.848;
   1:L PR[91] R[100]mm/sec CNT100;
   1:  PR[91,1] = PR[90,1] + 6.820;
   1:  PR[91,2] = PR[90,2] + 25.271;
   1:L PR[91] R[100]mm/sec CNT100;
   1:  PR[91,1] = PR[90,1] + 2.805;
   1:  PR[91,2] = PR[90,2] + 25.769;
   1:L PR[91] R[100]mm/sec CNT100;
   1:  PR[91,1] = PR[90,1] + 0.266;
   1:  PR[91,2] = PR[90,2] + 25.578;
   1:L PR[91] R[100]mm/sec CNT100;
   1:  PR[91] = PR[90];
   1:  PR[91,1] = PR[90,1] + -0.092;
   1:  PR[91,2] = PR[90,2] + 25.736;
   1:  PR[91,3] = PR[90,3] + 68.625;
   1:L PR[91] R[100]mm/sec CNT100;
   1:  PR[91,1] = PR[90,1] + -2.390;
   1:  PR[91,2] = PR[90,2] + 25.906;
   1:L PR[91] R[100]mm/sec CNT100;
   1:  PR[91,1] = PR[90,1] + -6.675;
   1:  PR[91,2] = PR[90,2] + 25.375;
   1:L PR[91] R[100]mm/sec CNT100;
   1:  PR[91,1] = PR[90,1] + -8.961;
   1:  PR[91,2] = PR[90,2] + 24.994;
   1:L PR[91] R[100]mm/sec CNT100;
   1:  PR[91,1] = PR[90,1] + -12.889;
   1:  PR[91,2] = PR[90,2] + 23.472;
   1:L PR[91] R[100]mm/sec CNT100;
   1:  PR[91,1] = PR[90,1] + -15.085;
   1:  PR[91,2] = PR[90,2] + 22.498;
   1:L PR[91] R[100]mm/sec CNT100;
   1:  PR[91,1] = PR[90,1] + -18.448;
   1:  PR[91,2] = PR[90,2] + 20.117;
   1:L PR[91] R[100]mm/sec CNT100;
   1:  PR[91,1] = PR[90,1] + -20.400;
   1:  PR[91,2] = PR[90,2] + 18.570;
   1:L PR[91] R[100]mm/sec CNT100;
   1:  PR[91,1] = PR[90,1] + -22.619;
   1:  PR[91,2] = PR[90,2] + 16.084;
   1:L PR[91] R[100]mm/sec CNT100;
   1:  PR[91,1] = PR[90,1] + -24.160;
   1:  PR[91,2] = PR[90,2] + 14.037;
   1:L PR[91] R[100]mm/sec CNT100;
   1:  PR[91,1] = PR[90,1] + -25.748;
   1:  PR[91,2] = PR[90,2] + 11.314;
   1:L PR[91] R[100]mm/sec CNT100;
   1:  PR[91,1] = PR[90,1] + -26.729;
   1:  PR[91,2] = PR[90,2] + 8.924;
   1:L PR[91] R[100]mm/sec CNT100;
   1:  PR[91,1] = PR[90,1] + -27.794;
   1:  PR[91,2] = PR[90,2] + 5.767;
   1:L PR[91] R[100]mm/sec CNT100;
   1:  PR[91,1] = PR[90,1] + -28.130;
   1:  PR[91,2] = PR[90,2] + 3.188;
   1:L PR[91] R[100]mm/sec CNT100;
   1:  PR[91,1] = PR[90,1] + -28.516;
   1:  PR[91,2] = PR[90,2] + -0.298;
   1:L PR[91] R[100]mm/sec CNT100;
   1:  PR[91,1] = PR[90,1] + -28.184;
   1:  PR[91,2] = PR[90,2] + -2.847;
   1:L PR[91] R[100]mm/sec CNT100;
   1:  PR[91,1] = PR[90,1] + -27.833;
   1:  PR[91,2] = PR[90,2] + -6.208;
   1:L PR[91] R[100]mm/sec CNT100;
   1:  PR[91,1] = PR[90,1] + -26.872;
   1:  PR[91,2] = PR[90,2] + -9.231;
   1:L PR[91] R[100]mm/sec CNT100;
   1:  PR[91,1] = PR[90,1] + -25.890;
   1:  PR[91,2] = PR[90,2] + -11.618;
   1:L PR[91] R[100]mm/sec CNT100;
   1:  PR[91,1] = PR[90,1] + -24.299;
   1:  PR[91,2] = PR[90,2] + -14.466;
   1:L PR[91] R[100]mm/sec CNT100;
   1:  PR[91,1] = PR[90,1] + -22.763;
   1:  PR[91,2] = PR[90,2] + -16.503;
   1:L PR[91] R[100]mm/sec CNT100;
   1:  PR[91,1] = PR[90,1] + -20.390;
   1:  PR[91,2] = PR[90,2] + -19.204;
   1:L PR[91] R[100]mm/sec CNT100;
   1:  PR[91,1] = PR[90,1] + -16.718;
   1:  PR[91,2] = PR[90,2] + -22.122;
   1:L PR[91] R[100]mm/sec CNT100;
   1:  PR[91,1] = PR[90,1] + -14.983;
   1:  PR[91,2] = PR[90,2] + -23.178;
   1:L PR[91] R[100]mm/sec CNT100;
   1:  PR[91,1] = PR[90,1] + -12.771;
   1:  PR[91,2] = PR[90,2] + -24.157;
   1:L PR[91] R[100]mm/sec CNT100;
   1:  PR[91,1] = PR[90,1] + -8.827;
   1:  PR[91,2] = PR[90,2] + -25.648;
   1:L PR[91] R[100]mm/sec CNT100;
   1:  PR[91,1] = PR[90,1] + -6.599;
   1:  PR[91,2] = PR[90,2] + -26.016;
   1:L PR[91] R[100]mm/sec CNT100;
   1:  PR[91,1] = PR[90,1] + -2.291;
   1:  PR[91,2] = PR[90,2] + -26.524;
   1:L PR[91] R[100]mm/sec CNT100;
   1:  PR[91,1] = PR[90,1] + -0.100;
   1:  PR[91,2] = PR[90,2] + -26.354;
   1:L PR[91] R[100]mm/sec CNT100;
   1:  PR[91,1] = PR[90,1] + 0.256;
   1:L PR[91] R[100]mm/sec CNT100;
   1:  PR[91,1] = PR[90,1] + 2.490;
   1:  PR[91,2] = PR[90,2] + -26.527;
   1:L PR[91] R[100]mm/sec CNT100;
   1:  PR[91,1] = PR[90,1] + 4.700;
   1:  PR[91,2] = PR[90,2] + -26.395;
   1:L PR[91] R[100]mm/sec CNT100;
   1:  PR[91,1] = PR[90,1] + 7.039;
   1:  PR[91,2] = PR[90,2] + -26.007;
   1:L PR[91] R[100]mm/sec CNT100;
   1:  PR[91,1] = PR[90,1] + 9.138;
   1:  PR[91,2] = PR[90,2] + -25.611;
   1:L PR[91] R[100]mm/sec CNT100;
   1:  PR[91,1] = PR[90,1] + 13.058;
   1:  PR[91,2] = PR[90,2] + -24.087;
   1:L PR[91] R[100]mm/sec CNT100;
   1:  PR[91,1] = PR[90,1] + 15.230;
   1:  PR[91,2] = PR[90,2] + -23.127;
   1:L PR[91] R[100]mm/sec CNT100;
   1:  PR[91,1] = PR[90,1] + 18.598;
   1:  PR[91,2] = PR[90,2] + -20.745;
   1:L PR[91] R[100]mm/sec CNT100;
   1:  PR[91,1] = PR[90,1] + 20.553;
   1:  PR[91,2] = PR[90,2] + -19.198;
   1:L PR[91] R[100]mm/sec CNT100;
   1:  PR[91,1] = PR[90,1] + 22.771;
   1:  PR[91,2] = PR[90,2] + -16.712;
   1:L PR[91] R[100]mm/sec CNT100;
   1:  PR[91,1] = PR[90,1] + 24.315;
   1:  PR[91,2] = PR[90,2] + -14.663;
   1:L PR[91] R[100]mm/sec CNT100;
   1:  PR[91,1] = PR[90,1] + 25.903;
   1:  PR[91,2] = PR[90,2] + -11.940;
   1:L PR[91] R[100]mm/sec CNT100;
   1:  PR[91,1] = PR[90,1] + 26.886;
   1:  PR[91,2] = PR[90,2] + -9.552;
   1:L PR[91] R[100]mm/sec CNT100;
   1:  PR[91,1] = PR[90,1] + 27.950;
   1:  PR[91,2] = PR[90,2] + -6.395;
   1:L PR[91] R[100]mm/sec CNT100;
   1:  PR[91,1] = PR[90,1] + 28.287;
   1:  PR[91,2] = PR[90,2] + -3.812;
   1:L PR[91] R[100]mm/sec CNT100;
   1:  PR[91,1] = PR[90,1] + 28.673;
   1:  PR[91,2] = PR[90,2] + -0.326;
   1:L PR[91] R[100]mm/sec CNT100;
   1:  PR[91,1] = PR[90,1] + 28.341;
   1:  PR[91,2] = PR[90,2] + 2.223;
   1:L PR[91] R[100]mm/sec CNT100;
   1:  PR[91,1] = PR[90,1] + 27.991;
   1:  PR[91,2] = PR[90,2] + 5.583;
   1:L PR[91] R[100]mm/sec CNT100;
   1:  PR[91,1] = PR[90,1] + 27.030;
   1:  PR[91,2] = PR[90,2] + 8.605;
   1:L PR[91] R[100]mm/sec CNT100;
   1:  PR[91,1] = PR[90,1] + 26.050;
   1:  PR[91,2] = PR[90,2] + 10.988;
   1:L PR[91] R[100]mm/sec CNT100;
   1:  PR[91,1] = PR[90,1] + 24.458;
   1:  PR[91,2] = PR[90,2] + 13.836;
   1:L PR[91] R[100]mm/sec CNT100;
   1:  PR[91,1] = PR[90,1] + 22.926;
   1:  PR[91,2] = PR[90,2] + 15.873;
   1:L PR[91] R[100]mm/sec CNT100;
   1:  PR[91,1] = PR[90,1] + 20.554;
   1:  PR[91,2] = PR[90,2] + 18.573;
   1:L PR[91] R[100]mm/sec CNT100;
   1:  PR[91,1] = PR[90,1] + 18.605;
   1:  PR[91,2] = PR[90,2] + 20.117;
   1:L PR[91] R[100]mm/sec CNT100;
   1:  PR[91,1] = PR[90,1] + 15.243;
   1:  PR[91,2] = PR[90,2] + 22.498;
   1:L PR[91] R[100]mm/sec CNT100;
   1:  PR[91,1] = PR[90,1] + 13.047;
   1:  PR[91,2] = PR[90,2] + 23.472;
   1:L PR[91] R[100]mm/sec CNT100;
   1:  PR[91,1] = PR[90,1] + 9.117;
   1:  PR[91,2] = PR[90,2] + 24.994;
   1:L PR[91] R[100]mm/sec CNT100;
   1:  PR[91,1] = PR[90,1] + 6.832;
   1:  PR[91,2] = PR[90,2] + 25.375;
   1:L PR[91] R[100]mm/sec CNT100;
   1:  PR[91,1] = PR[90,1] + 2.546;
   1:  PR[91,2] = PR[90,2] + 25.906;
   1:L PR[91] R[100]mm/sec CNT100;
   1:  PR[91,1] = PR[90,1] + 0.252;
   1:  PR[91,2] = PR[90,2] + 25.736;
   1:L PR[91] R[100]mm/sec CNT100;
   1:  PR[91] = PR[90];
   1:  PR[91,1] = PR[90,1] + -0.083;
   1:  PR[91,2] = PR[90,2] + 25.892;
   1:  PR[91,3] = PR[90,3] + 69.235;
   1:L PR[91] R[100]mm/sec CNT100;
   1:  PR[91,1] = PR[90,1] + -2.132;
   1:  PR[91,2] = PR[90,2] + 26.044;
   1:L PR[91] R[100]mm/sec CNT100;
   1:  PR[91,1] = PR[90,1] + -6.687;
   1:  PR[91,2] = PR[90,2] + 25.479;
   1:L PR[91] R[100]mm/sec CNT100;
   1:  PR[91,1] = PR[90,1] + -8.719;
   1:  PR[91,2] = PR[90,2] + 25.141;
   1:L PR[91] R[100]mm/sec CNT100;
   1:  PR[91,1] = PR[90,1] + -12.910;
   1:  PR[91,2] = PR[90,2] + 23.517;
   1:L PR[91] R[100]mm/sec CNT100;
   1:  PR[91,1] = PR[90,1] + -14.863;
   1:  PR[91,2] = PR[90,2] + 22.650;
   1:L PR[91] R[100]mm/sec CNT100;
   1:  PR[91,1] = PR[90,1] + -18.463;
   1:  PR[91,2] = PR[90,2] + 20.101;
   1:L PR[91] R[100]mm/sec CNT100;
   1:  PR[91,1] = PR[90,1] + -20.201;
   1:  PR[91,2] = PR[90,2] + 18.724;
   1:L PR[91] R[100]mm/sec CNT100;
   1:  PR[91,1] = PR[90,1] + -22.586;
   1:  PR[91,2] = PR[90,2] + 16.051;
   1:L PR[91] R[100]mm/sec CNT100;
   1:  PR[91,1] = PR[90,1] + -23.957;
   1:  PR[91,2] = PR[90,2] + 14.230;
   1:L PR[91] R[100]mm/sec CNT100;
   1:  PR[91,1] = PR[90,1] + -25.670;
   1:  PR[91,2] = PR[90,2] + 11.294;
   1:L PR[91] R[100]mm/sec CNT100;
   1:  PR[91,1] = PR[90,1] + -26.542;
   1:  PR[91,2] = PR[90,2] + 9.171;
   1:L PR[91] R[100]mm/sec CNT100;
   1:  PR[91,1] = PR[90,1] + -27.692;
   1:  PR[91,2] = PR[90,2] + 5.760;
   1:L PR[91] R[100]mm/sec CNT100;
   1:  PR[91,1] = PR[90,1] + -27.990;
   1:  PR[91,2] = PR[90,2] + 3.472;
   1:L PR[91] R[100]mm/sec CNT100;
   1:  PR[91,1] = PR[90,1] + -28.408;
   1:  PR[91,2] = PR[90,2] + -0.298;
   1:L PR[91] R[100]mm/sec CNT100;
   1:  PR[91,1] = PR[90,1] + -28.113;
   1:  PR[91,2] = PR[90,2] + -2.558;
   1:L PR[91] R[100]mm/sec CNT100;
   1:  PR[91,1] = PR[90,1] + -27.735;
   1:  PR[91,2] = PR[90,2] + -6.185;
   1:L PR[91] R[100]mm/sec CNT100;
   1:  PR[91,1] = PR[90,1] + -26.696;
   1:  PR[91,2] = PR[90,2] + -9.452;
   1:L PR[91] R[100]mm/sec CNT100;
   1:  PR[91,1] = PR[90,1] + -25.824;
   1:  PR[91,2] = PR[90,2] + -11.573;
   1:L PR[91] R[100]mm/sec CNT100;
   1:  PR[91,1] = PR[90,1] + -24.108;
   1:  PR[91,2] = PR[90,2] + -14.643;
   1:L PR[91] R[100]mm/sec CNT100;
   1:  PR[91,1] = PR[90,1] + -22.742;
   1:  PR[91,2] = PR[90,2] + -16.454;
   1:L PR[91] R[100]mm/sec CNT100;
   1:  PR[91,1] = PR[90,1] + -20.191;
   1:  PR[91,2] = PR[90,2] + -19.357;
   1:L PR[91] R[100]mm/sec CNT100;
   1:  PR[91,1] = PR[90,1] + -16.615;
   1:  PR[91,2] = PR[90,2] + -22.201;
   1:L PR[91] R[100]mm/sec CNT100;
   1:  PR[91,1] = PR[90,1] + -14.753;
   1:  PR[91,2] = PR[90,2] + -23.335;
   1:L PR[91] R[100]mm/sec CNT100;
   1:  PR[91,1] = PR[90,1] + -12.786;
   1:  PR[91,2] = PR[90,2] + -24.205;
   1:L PR[91] R[100]mm/sec CNT100;
   1:  PR[91,1] = PR[90,1] + -8.578;
   1:  PR[91,2] = PR[90,2] + -25.796;
   1:L PR[91] R[100]mm/sec CNT100;
   1:  PR[91,1] = PR[90,1] + -6.608;
   1:  PR[91,2] = PR[90,2] + -26.121;
   1:L PR[91] R[100]mm/sec CNT100;
   1:  PR[91,1] = PR[90,1] + -2.029;
   1:  PR[91,2] = PR[90,2] + -26.661;
   1:L PR[91] R[100]mm/sec CNT100;
   1:  PR[91,1] = PR[90,1] + -0.087;
   1:  PR[91,2] = PR[90,2] + -26.510;
   1:L PR[91] R[100]mm/sec CNT100;
   1:  PR[91,1] = PR[90,1] + 0.244;
   1:L PR[91] R[100]mm/sec CNT100;
   1:  PR[91,1] = PR[90,1] + 2.228;
   1:  PR[91,2] = PR[90,2] + -26.664;
   1:L PR[91] R[100]mm/sec CNT100;
   1:  PR[91,1] = PR[90,1] + 4.582;
   1:  PR[91,2] = PR[90,2] + -26.524;
   1:L PR[91] R[100]mm/sec CNT100;
   1:  PR[91,1] = PR[90,1] + 6.658;
   1:  PR[91,2] = PR[90,2] + -26.179;
   1:L PR[91] R[100]mm/sec CNT100;
   1:  PR[91,1] = PR[90,1] + 8.901;
   1:  PR[91,2] = PR[90,2] + -25.756;
   1:L PR[91] R[100]mm/sec CNT100;
   1:  PR[91,1] = PR[90,1] + 13.082;
   1:  PR[91,2] = PR[90,2] + -24.130;
   1:L PR[91] R[100]mm/sec CNT100;
   1:  PR[91,1] = PR[90,1] + 15.008;
   1:  PR[91,2] = PR[90,2] + -23.279;
   1:L PR[91] R[100]mm/sec CNT100;
   1:  PR[91,1] = PR[90,1] + 18.614;
   1:  PR[91,2] = PR[90,2] + -20.729;
   1:L PR[91] R[100]mm/sec CNT100;
   1:  PR[91,1] = PR[90,1] + 20.355;
   1:  PR[91,2] = PR[90,2] + -19.352;
   1:L PR[91] R[100]mm/sec CNT100;
